  [1553] = {x=-964.119, y=28.121, z=22, rx=180, rz=142.037, shoulder=lefty, elbow=epositive, wrist=wpositive, fatherId=fReference[0]}
  [1554] = {x=-962.88, y=29.088, z=22, rx=180, rz=142.05, shoulder=lefty, elbow=epositive, wrist=wpositive, fatherId=fReference[0]}
  [1555] = {x=-961.641, y=30.054, z=22, rx=180, rz=142.063, shoulder=lefty, elbow=epositive, wrist=wpositive, fatherId=fReference[0]}
  [1556] = {x=-960.402, y=31.02, z=22, rx=180, rz=142.076, shoulder=lefty, elbow=epositive, wrist=wpositive, fatherId=fReference[0]}
  [1557] = {x=-959.163, y=31.986, z=22, rx=180, rz=142.09, shoulder=lefty, elbow=epositive, wrist=wpositive, fatherId=fReference[0]}
  [1558] = {x=-957.923, y=32.951, z=22, rx=180, rz=142.105, shoulder=lefty, elbow=epositive, wrist=wpositive, fatherId=fReference[0]}
  [1559] = {x=-956.684, y=33.916, z=22, rx=180, rz=142.12, shoulder=lefty, elbow=epositive, wrist=wpositive, fatherId=fReference[0]}
  [1560] = {x=-955.444, y=34.88, z=22, rx=180, rz=142.135, shoulder=lefty, elbow=epositive, wrist=wpositive, fatherId=fReference[0]}
  [1561] = {x=-954.204, y=35.844, z=22, rx=180, rz=142.151, shoulder=lefty, elbow=epositive, wrist=wpositive, fatherId=fReference[0]}
  [1562] = {x=-952.964, y=36.808, z=22, rx=180, rz=142.167, shoulder=lefty, elbow=epositive, wrist=wpositive, fatherId=fReference[0]}
  [1563] = {x=-951.724, y=37.771, z=22, rx=180, rz=142.183, shoulder=lefty, elbow=epositive, wrist=wpositive, fatherId=fReference[0]}
  [1564] = {x=-950.483, y=38.734, z=22, rx=180, rz=142.2, shoulder=lefty, elbow=epositive, wrist=wpositive, fatherId=fReference[0]}
  [1565] = {x=-949.243, y=39.696, z=22, rx=180, rz=142.218, shoulder=lefty, elbow=epositive, wrist=wpositive, fatherId=fReference[0]}
  [1566] = {x=-948.002, y=40.658, z=22, rx=180, rz=142.235, shoulder=lefty, elbow=epositive, wrist=wpositive, fatherId=fReference[0]}
  [1567] = {x=-946.761, y=41.619, z=22, rx=180, rz=142.254, shoulder=lefty, elbow=epositive, wrist=wpositive, fatherId=fReference[0]}
  [1568] = {x=-945.52, y=42.58, z=22, rx=180, rz=142.272, shoulder=lefty, elbow=epositive, wrist=wpositive, fatherId=fReference[0]}
  [1569] = {x=-944.278, y=43.541, z=22, rx=180, rz=142.291, shoulder=lefty, elbow=epositive, wrist=wpositive, fatherId=fReference[0]}
  [1570] = {x=-943.037, y=44.501, z=22, rx=180, rz=142.311, shoulder=lefty, elbow=epositive, wrist=wpositive, fatherId=fReference[0]}
  [1571] = {x=-941.795, y=45.46, z=22, rx=180, rz=142.331, shoulder=lefty, elbow=epositive, wrist=wpositive, fatherId=fReference[0]}
  [1572] = {x=-940.553, y=46.419, z=22, rx=180, rz=142.351, shoulder=lefty, elbow=epositive, wrist=wpositive, fatherId=fReference[0]}
  [1573] = {x=-939.31, y=47.377, z=22, rx=180, rz=142.372, shoulder=lefty, elbow=epositive, wrist=wpositive, fatherId=fReference[0]}
  [1574] = {x=-938.068, y=48.335, z=22, rx=180, rz=142.394, shoulder=lefty, elbow=epositive, wrist=wpositive, fatherId=fReference[0]}
  [1575] = {x=-936.825, y=49.292, z=22, rx=180, rz=142.415, shoulder=lefty, elbow=epositive, wrist=wpositive, fatherId=fReference[0]}
  [1576] = {x=-935.582, y=50.249, z=22, rx=180, rz=142.438, shoulder=lefty, elbow=epositive, wrist=wpositive, fatherId=fReference[0]}
  [1577] = {x=-934.339, y=51.205, z=22, rx=180, rz=142.46, shoulder=lefty, elbow=epositive, wrist=wpositive, fatherId=fReference[0]}
  [1578] = {x=-933.095, y=52.161, z=22, rx=180, rz=142.483, shoulder=lefty, elbow=epositive, wrist=wpositive, fatherId=fReference[0]}
  [1579] = {x=-931.852, y=53.116, z=22, rx=180, rz=142.507, shoulder=lefty, elbow=epositive, wrist=wpositive, fatherId=fReference[0]}
  [1580] = {x=-930.608, y=54.07, z=22, rx=180, rz=142.531, shoulder=lefty, elbow=epositive, wrist=wpositive, fatherId=fReference[0]}
  [1581] = {x=-929.363, y=55.024, z=22, rx=180, rz=142.555, shoulder=lefty, elbow=epositive, wrist=wpositive, fatherId=fReference[0]}
  [1582] = {x=-928.119, y=55.977, z=22, rx=180, rz=142.58, shoulder=lefty, elbow=epositive, wrist=wpositive, fatherId=fReference[0]}
  [1583] = {x=-926.874, y=56.929, z=22, rx=180, rz=142.605, shoulder=lefty, elbow=epositive, wrist=wpositive, fatherId=fReference[0]}
  [1584] = {x=-925.629, y=57.881, z=22, rx=180, rz=142.631, shoulder=lefty, elbow=epositive, wrist=wpositive, fatherId=fReference[0]}
  [1585] = {x=-924.384, y=58.832, z=22, rx=180, rz=142.657, shoulder=lefty, elbow=epositive, wrist=wpositive, fatherId=fReference[0]}
  [1586] = {x=-923.138, y=59.782, z=22, rx=180, rz=142.684, shoulder=lefty, elbow=epositive, wrist=wpositive, fatherId=fReference[0]}
  [1587] = {x=-921.892, y=60.732, z=22, rx=180, rz=142.711, shoulder=lefty, elbow=epositive, wrist=wpositive, fatherId=fReference[0]}
  [1588] = {x=-920.646, y=61.681, z=22, rx=180, rz=142.738, shoulder=lefty, elbow=epositive, wrist=wpositive, fatherId=fReference[0]}
  [1589] = {x=-919.4, y=62.629, z=22, rx=180, rz=142.766, shoulder=lefty, elbow=epositive, wrist=wpositive, fatherId=fReference[0]}
  [1590] = {x=-918.153, y=63.576, z=22, rx=180, rz=142.795, shoulder=lefty, elbow=epositive, wrist=wpositive, fatherId=fReference[0]}
  [1591] = {x=-916.906, y=64.523, z=22, rx=180, rz=142.824, shoulder=lefty, elbow=epositive, wrist=wpositive, fatherId=fReference[0]}
  [1592] = {x=-915.659, y=65.469, z=22, rx=180, rz=142.853, shoulder=lefty, elbow=epositive, wrist=wpositive, fatherId=fReference[0]}
  [1593] = {x=-914.411, y=66.414, z=22, rx=180, rz=142.883, shoulder=lefty, elbow=epositive, wrist=wpositive, fatherId=fReference[0]}
  [1594] = {x=-913.163, y=67.358, z=22, rx=180, rz=142.913, shoulder=lefty, elbow=epositive, wrist=wpositive, fatherId=fReference[0]}
  [1595] = {x=-911.915, y=68.302, z=22, rx=180, rz=142.944, shoulder=lefty, elbow=epositive, wrist=wpositive, fatherId=fReference[0]}
  [1596] = {x=-910.667, y=69.245, z=22, rx=180, rz=142.975, shoulder=lefty, elbow=epositive, wrist=wpositive, fatherId=fReference[0]}
  [1597] = {x=-909.418, y=70.187, z=22, rx=180, rz=143.007, shoulder=lefty, elbow=epositive, wrist=wpositive, fatherId=fReference[0]}
  [1598] = {x=-908.169, y=71.128, z=22, rx=180, rz=143.039, shoulder=lefty, elbow=epositive, wrist=wpositive, fatherId=fReference[0]}
  [1599] = {x=-906.919, y=72.068, z=22, rx=180, rz=143.071, shoulder=lefty, elbow=epositive, wrist=wpositive, fatherId=fReference[0]}
  [1600] = {x=-905.67, y=73.007, z=22, rx=180, rz=143.104, shoulder=lefty, elbow=epositive, wrist=wpositive, fatherId=fReference[0]}
  [1601] = {x=-904.419, y=73.946, z=22, rx=180, rz=143.138, shoulder=lefty, elbow=epositive, wrist=wpositive, fatherId=fReference[0]}
  [1602] = {x=-903.169, y=74.883, z=22, rx=180, rz=143.172, shoulder=lefty, elbow=epositive, wrist=wpositive, fatherId=fReference[0]}
  [1603] = {x=-901.918, y=75.82, z=22, rx=180, rz=143.206, shoulder=lefty, elbow=epositive, wrist=wpositive, fatherId=fReference[0]}
  [1604] = {x=-900.667, y=76.756, z=22, rx=180, rz=143.241, shoulder=lefty, elbow=epositive, wrist=wpositive, fatherId=fReference[0]}
  [1605] = {x=-899.416, y=77.691, z=22, rx=180, rz=143.276, shoulder=lefty, elbow=epositive, wrist=wpositive, fatherId=fReference[0]}
  [1606] = {x=-898.164, y=78.625, z=22, rx=180, rz=143.312, shoulder=lefty, elbow=epositive, wrist=wpositive, fatherId=fReference[0]}
  [1607] = {x=-896.912, y=79.557, z=22, rx=180, rz=143.348, shoulder=lefty, elbow=epositive, wrist=wpositive, fatherId=fReference[0]}
  [1608] = {x=-895.659, y=80.489, z=22, rx=180, rz=143.385, shoulder=lefty, elbow=epositive, wrist=wpositive, fatherId=fReference[0]}
  [1609] = {x=-894.406, y=81.42, z=22, rx=180, rz=143.422, shoulder=lefty, elbow=epositive, wrist=wpositive, fatherId=fReference[0]}
  [1610] = {x=-893.153, y=82.35, z=22, rx=180, rz=143.46, shoulder=lefty, elbow=epositive, wrist=wpositive, fatherId=fReference[0]}
  [1611] = {x=-891.899, y=83.279, z=22, rx=180, rz=143.498, shoulder=lefty, elbow=epositive, wrist=wpositive, fatherId=fReference[0]}
  [1612] = {x=-890.645, y=84.207, z=22, rx=180, rz=143.536, shoulder=lefty, elbow=epositive, wrist=wpositive, fatherId=fReference[0]}
  [1613] = {x=-889.391, y=85.134, z=22, rx=180, rz=143.575, shoulder=lefty, elbow=epositive, wrist=wpositive, fatherId=fReference[0]}
  [1614] = {x=-888.136, y=86.06, z=22, rx=180, rz=143.615, shoulder=lefty, elbow=epositive, wrist=wpositive, fatherId=fReference[0]}
  [1615] = {x=-886.881, y=86.985, z=22, rx=180, rz=143.655, shoulder=lefty, elbow=epositive, wrist=wpositive, fatherId=fReference[0]}
  [1616] = {x=-885.626, y=87.909, z=22, rx=180, rz=143.696, shoulder=lefty, elbow=epositive, wrist=wpositive, fatherId=fReference[0]}
  [1617] = {x=-884.37, y=88.832, z=22, rx=180, rz=143.737, shoulder=lefty, elbow=epositive, wrist=wpositive, fatherId=fReference[0]}
  [1618] = {x=-883.113, y=89.753, z=22, rx=180, rz=143.778, shoulder=lefty, elbow=epositive, wrist=wpositive, fatherId=fReference[0]}
  [1619] = {x=-881.857, y=90.674, z=22, rx=180, rz=143.82, shoulder=lefty, elbow=epositive, wrist=wpositive, fatherId=fReference[0]}
  [1620] = {x=-880.6, y=91.593, z=22, rx=180, rz=143.862, shoulder=lefty, elbow=epositive, wrist=wpositive, fatherId=fReference[0]}
  [1621] = {x=-879.342, y=92.511, z=22, rx=180, rz=143.905, shoulder=lefty, elbow=epositive, wrist=wpositive, fatherId=fReference[0]}
  [1622] = {x=-878.084, y=93.428, z=22, rx=180, rz=143.949, shoulder=lefty, elbow=epositive, wrist=wpositive, fatherId=fReference[0]}
  [1623] = {x=-876.826, y=94.344, z=22, rx=180, rz=143.993, shoulder=lefty, elbow=epositive, wrist=wpositive, fatherId=fReference[0]}
  [1624] = {x=-875.567, y=95.259, z=22, rx=180, rz=144.037, shoulder=lefty, elbow=epositive, wrist=wpositive, fatherId=fReference[0]}
  [1625] = {x=-874.308, y=96.173, z=22, rx=180, rz=144.082, shoulder=lefty, elbow=epositive, wrist=wpositive, fatherId=fReference[0]}
  [1626] = {x=-873.049, y=97.085, z=22, rx=180, rz=144.127, shoulder=lefty, elbow=epositive, wrist=wpositive, fatherId=fReference[0]}
  [1627] = {x=-871.789, y=97.996, z=22, rx=180, rz=144.173, shoulder=lefty, elbow=epositive, wrist=wpositive, fatherId=fReference[0]}
  [1628] = {x=-870.528, y=98.906, z=22, rx=-180, rz=144.22, shoulder=lefty, elbow=epositive, wrist=wpositive, fatherId=fReference[0]}
  [1629] = {x=-869.267, y=99.815, z=22, rx=180, rz=144.266, shoulder=lefty, elbow=epositive, wrist=wpositive, fatherId=fReference[0]}
  [1630] = {x=-868.006, y=100.722, z=22, rx=180, rz=144.314, shoulder=lefty, elbow=epositive, wrist=wpositive, fatherId=fReference[0]}
  [1631] = {x=-866.745, y=101.628, z=22, rx=180, rz=144.362, shoulder=lefty, elbow=epositive, wrist=wpositive, fatherId=fReference[0]}
  [1632] = {x=-865.482, y=102.533, z=22, rx=180, rz=144.41, shoulder=lefty, elbow=epositive, wrist=wpositive, fatherId=fReference[0]}
  [1633] = {x=-864.22, y=103.437, z=22, rx=180, rz=144.459, shoulder=lefty, elbow=epositive, wrist=wpositive, fatherId=fReference[0]}
  [1634] = {x=-862.957, y=104.339, z=22, rx=180, rz=144.508, shoulder=lefty, elbow=epositive, wrist=wpositive, fatherId=fReference[0]}
  [1635] = {x=-861.693, y=105.24, z=22, rx=180, rz=144.558, shoulder=lefty, elbow=epositive, wrist=wpositive, fatherId=fReference[0]}
  [1636] = {x=-860.429, y=106.139, z=22, rx=180, rz=144.609, shoulder=lefty, elbow=epositive, wrist=wpositive, fatherId=fReference[0]}
  [1637] = {x=-859.165, y=107.038, z=22, rx=180, rz=144.659, shoulder=lefty, elbow=epositive, wrist=wpositive, fatherId=fReference[0]}
  [1638] = {x=-857.9, y=107.935, z=22, rx=180, rz=144.711, shoulder=lefty, elbow=epositive, wrist=wpositive, fatherId=fReference[0]}
  [1639] = {x=-856.635, y=108.83, z=22, rx=180, rz=144.763, shoulder=lefty, elbow=epositive, wrist=wpositive, fatherId=fReference[0]}
  [1640] = {x=-855.369, y=109.724, z=22, rx=180, rz=144.815, shoulder=lefty, elbow=epositive, wrist=wpositive, fatherId=fReference[0]}
  [1641] = {x=-854.103, y=110.617, z=22, rx=180, rz=144.868, shoulder=lefty, elbow=epositive, wrist=wpositive, fatherId=fReference[0]}
  [1642] = {x=-852.836, y=111.508, z=22, rx=180, rz=144.922, shoulder=lefty, elbow=epositive, wrist=wpositive, fatherId=fReference[0]}
  [1643] = {x=-851.569, y=112.398, z=22, rx=180, rz=144.976, shoulder=lefty, elbow=epositive, wrist=wpositive, fatherId=fReference[0]}
  [1644] = {x=-850.301, y=113.287, z=22, rx=180, rz=145.03, shoulder=lefty, elbow=epositive, wrist=wpositive, fatherId=fReference[0]}
  [1645] = {x=-849.033, y=114.174, z=22, rx=180, rz=145.085, shoulder=lefty, elbow=epositive, wrist=wpositive, fatherId=fReference[0]}
  [1646] = {x=-847.764, y=115.059, z=22, rx=180, rz=145.141, shoulder=lefty, elbow=epositive, wrist=wpositive, fatherId=fReference[0]}
  [1647] = {x=-846.495, y=115.943, z=22, rx=180, rz=145.197, shoulder=lefty, elbow=epositive, wrist=wpositive, fatherId=fReference[0]}
  [1648] = {x=-845.225, y=116.826, z=22, rx=180, rz=145.253, shoulder=lefty, elbow=epositive, wrist=wpositive, fatherId=fReference[0]}
  [1649] = {x=-843.955, y=117.707, z=22, rx=180, rz=145.311, shoulder=lefty, elbow=epositive, wrist=wpositive, fatherId=fReference[0]}
  [1650] = {x=-842.685, y=118.586, z=22, rx=180, rz=145.368, shoulder=lefty, elbow=epositive, wrist=wpositive, fatherId=fReference[0]}
  [1651] = {x=-841.413, y=119.464, z=22, rx=180, rz=145.426, shoulder=lefty, elbow=epositive, wrist=wpositive, fatherId=fReference[0]}
  [1652] = {x=-840.142, y=120.341, z=22, rx=180, rz=145.485, shoulder=lefty, elbow=epositive, wrist=wpositive, fatherId=fReference[0]}
  [1653] = {x=-838.869, y=121.216, z=22, rx=180, rz=145.544, shoulder=lefty, elbow=epositive, wrist=wpositive, fatherId=fReference[0]}
  [1654] = {x=-837.597, y=122.089, z=22, rx=180, rz=145.604, shoulder=lefty, elbow=epositive, wrist=wpositive, fatherId=fReference[0]}
  [1655] = {x=-836.323, y=122.961, z=22, rx=180, rz=145.665, shoulder=lefty, elbow=epositive, wrist=wpositive, fatherId=fReference[0]}
  [1656] = {x=-835.049, y=123.831, z=22, rx=180, rz=145.725, shoulder=lefty, elbow=epositive, wrist=wpositive, fatherId=fReference[0]}
  [1657] = {x=-833.775, y=124.699, z=22, rx=180, rz=145.787, shoulder=lefty, elbow=epositive, wrist=wpositive, fatherId=fReference[0]}
  [1658] = {x=-832.5, y=125.566, z=22, rx=-180, rz=145.849, shoulder=lefty, elbow=epositive, wrist=wpositive, fatherId=fReference[0]}
  [1659] = {x=-831.225, y=126.431, z=22, rx=180, rz=145.911, shoulder=lefty, elbow=epositive, wrist=wpositive, fatherId=fReference[0]}
  [1660] = {x=-829.949, y=127.295, z=22, rx=180, rz=145.974, shoulder=lefty, elbow=epositive, wrist=wpositive, fatherId=fReference[0]}
  [1661] = {x=-828.672, y=128.157, z=22, rx=180, rz=146.038, shoulder=lefty, elbow=epositive, wrist=wpositive, fatherId=fReference[0]}
  [1662] = {x=-827.395, y=129.017, z=22, rx=180, rz=146.102, shoulder=lefty, elbow=epositive, wrist=wpositive, fatherId=fReference[0]}
  [1663] = {x=-826.117, y=129.876, z=22, rx=180, rz=146.167, shoulder=lefty, elbow=epositive, wrist=wpositive, fatherId=fReference[0]}
  [1664] = {x=-824.839, y=130.732, z=22, rx=180, rz=146.232, shoulder=lefty, elbow=epositive, wrist=wpositive, fatherId=fReference[0]}
  [1665] = {x=-823.56, y=131.587, z=22, rx=180, rz=146.298, shoulder=lefty, elbow=epositive, wrist=wpositive, fatherId=fReference[0]}
  [1666] = {x=-822.281, y=132.441, z=22, rx=180, rz=146.364, shoulder=lefty, elbow=epositive, wrist=wpositive, fatherId=fReference[0]}
  [1667] = {x=-821.001, y=133.292, z=22, rx=180, rz=146.431, shoulder=lefty, elbow=epositive, wrist=wpositive, fatherId=fReference[0]}
  [1668] = {x=-819.721, y=134.142, z=22, rx=-180, rz=146.499, shoulder=lefty, elbow=epositive, wrist=wpositive, fatherId=fReference[0]}
  [1669] = {x=-818.44, y=134.99, z=22, rx=180, rz=146.567, shoulder=lefty, elbow=epositive, wrist=wpositive, fatherId=fReference[0]}
  [1670] = {x=-817.158, y=135.836, z=22, rx=180, rz=146.636, shoulder=lefty, elbow=epositive, wrist=wpositive, fatherId=fReference[0]}
  [1671] = {x=-815.876, y=136.68, z=22, rx=180, rz=146.705, shoulder=lefty, elbow=epositive, wrist=wpositive, fatherId=fReference[0]}
  [1672] = {x=-814.593, y=137.523, z=22, rx=180, rz=146.775, shoulder=lefty, elbow=epositive, wrist=wpositive, fatherId=fReference[0]}
  [1673] = {x=-813.309, y=138.364, z=22, rx=180, rz=146.845, shoulder=lefty, elbow=epositive, wrist=wpositive, fatherId=fReference[0]}
  [1674] = {x=-812.025, y=139.202, z=22, rx=180, rz=146.916, shoulder=lefty, elbow=epositive, wrist=wpositive, fatherId=fReference[0]}
  [1675] = {x=-810.74, y=140.039, z=22, rx=180, rz=146.987, shoulder=lefty, elbow=epositive, wrist=wpositive, fatherId=fReference[0]}
  [1676] = {x=-809.455, y=140.875, z=22, rx=180, rz=147.059, shoulder=lefty, elbow=epositive, wrist=wpositive, fatherId=fReference[0]}
  [1677] = {x=-808.169, y=141.708, z=22, rx=180, rz=147.132, shoulder=lefty, elbow=epositive, wrist=wpositive, fatherId=fReference[0]}
  [1678] = {x=-806.883, y=142.539, z=22, rx=180, rz=147.205, shoulder=lefty, elbow=epositive, wrist=wpositive, fatherId=fReference[0]}
  [1679] = {x=-805.596, y=143.368, z=22, rx=180, rz=147.279, shoulder=lefty, elbow=epositive, wrist=wpositive, fatherId=fReference[0]}
  [1680] = {x=-804.308, y=144.196, z=22, rx=180, rz=147.353, shoulder=lefty, elbow=epositive, wrist=wpositive, fatherId=fReference[0]}
  [1681] = {x=-803.019, y=145.021, z=22, rx=180, rz=147.428, shoulder=lefty, elbow=epositive, wrist=wpositive, fatherId=fReference[0]}
  [1682] = {x=-801.73, y=145.845, z=22, rx=-180, rz=147.504, shoulder=lefty, elbow=epositive, wrist=wpositive, fatherId=fReference[0]}
  [1683] = {x=-800.44, y=146.666, z=22, rx=180, rz=147.58, shoulder=lefty, elbow=epositive, wrist=wpositive, fatherId=fReference[0]}
  [1684] = {x=-799.15, y=147.486, z=22, rx=180, rz=147.657, shoulder=lefty, elbow=epositive, wrist=wpositive, fatherId=fReference[0]}
  [1685] = {x=-797.859, y=148.303, z=22, rx=180, rz=147.734, shoulder=lefty, elbow=epositive, wrist=wpositive, fatherId=fReference[0]}
  [1686] = {x=-796.567, y=149.119, z=22, rx=180, rz=147.812, shoulder=lefty, elbow=epositive, wrist=wpositive, fatherId=fReference[0]}
  [1687] = {x=-795.275, y=149.932, z=22, rx=180, rz=147.891, shoulder=lefty, elbow=epositive, wrist=wpositive, fatherId=fReference[0]}
  [1688] = {x=-793.982, y=150.744, z=22, rx=180, rz=147.97, shoulder=lefty, elbow=epositive, wrist=wpositive, fatherId=fReference[0]}
  [1689] = {x=-792.688, y=151.553, z=22, rx=-180, rz=148.05, shoulder=lefty, elbow=epositive, wrist=wpositive, fatherId=fReference[0]}
  [1690] = {x=-791.394, y=152.36, z=22, rx=180, rz=148.13, shoulder=lefty, elbow=epositive, wrist=wpositive, fatherId=fReference[0]}
  [1691] = {x=-790.099, y=153.165, z=22, rx=180, rz=148.211, shoulder=lefty, elbow=epositive, wrist=wpositive, fatherId=fReference[0]}
  [1692] = {x=-788.803, y=153.968, z=22, rx=-180, rz=148.293, shoulder=lefty, elbow=epositive, wrist=wpositive, fatherId=fReference[0]}
  [1693] = {x=-787.507, y=154.769, z=22, rx=180, rz=148.375, shoulder=lefty, elbow=epositive, wrist=wpositive, fatherId=fReference[0]}
  [1694] = {x=-786.21, y=155.568, z=22, rx=180, rz=148.458, shoulder=lefty, elbow=epositive, wrist=wpositive, fatherId=fReference[0]}
  [1695] = {x=-784.912, y=156.365, z=22, rx=180, rz=148.541, shoulder=lefty, elbow=epositive, wrist=wpositive, fatherId=fReference[0]}
  [1696] = {x=-783.613, y=157.159, z=22, rx=-180, rz=148.625, shoulder=lefty, elbow=epositive, wrist=wpositive, fatherId=fReference[0]}
  [1697] = {x=-782.314, y=157.951, z=22, rx=180, rz=148.71, shoulder=lefty, elbow=epositive, wrist=wpositive, fatherId=fReference[0]}
  [1698] = {x=-781.014, y=158.741, z=22, rx=180, rz=148.795, shoulder=lefty, elbow=epositive, wrist=wpositive, fatherId=fReference[0]}
  [1699] = {x=-779.714, y=159.529, z=22, rx=180, rz=148.881, shoulder=lefty, elbow=epositive, wrist=wpositive, fatherId=fReference[0]}
  [1700] = {x=-778.413, y=160.315, z=22, rx=180, rz=148.968, shoulder=lefty, elbow=epositive, wrist=wpositive, fatherId=fReference[0]}
  [1701] = {x=-777.111, y=161.098, z=22, rx=180, rz=149.055, shoulder=lefty, elbow=epositive, wrist=wpositive, fatherId=fReference[0]}
  [1702] = {x=-775.808, y=161.879, z=22, rx=180, rz=149.143, shoulder=lefty, elbow=epositive, wrist=wpositive, fatherId=fReference[0]}
  [1703] = {x=-774.505, y=162.658, z=22, rx=180, rz=149.231, shoulder=lefty, elbow=epositive, wrist=wpositive, fatherId=fReference[0]}
  [1704] = {x=-773.2, y=163.434, z=22, rx=-180, rz=149.32, shoulder=lefty, elbow=epositive, wrist=wpositive, fatherId=fReference[0]}
  [1705] = {x=-771.896, y=164.208, z=22, rx=180, rz=149.41, shoulder=lefty, elbow=epositive, wrist=wpositive, fatherId=fReference[0]}
  [1706] = {x=-770.59, y=164.98, z=22, rx=180, rz=149.5, shoulder=lefty, elbow=epositive, wrist=wpositive, fatherId=fReference[0]}
  [1707] = {x=-769.284, y=165.75, z=22, rx=180, rz=149.591, shoulder=lefty, elbow=epositive, wrist=wpositive, fatherId=fReference[0]}
  [1708] = {x=-767.977, y=166.517, z=22, rx=180, rz=149.683, shoulder=lefty, elbow=epositive, wrist=wpositive, fatherId=fReference[0]}
  [1709] = {x=-766.669, y=167.281, z=22, rx=180, rz=149.775, shoulder=lefty, elbow=epositive, wrist=wpositive, fatherId=fReference[0]}
  [1710] = {x=-765.36, y=168.044, z=22, rx=180, rz=149.868, shoulder=lefty, elbow=epositive, wrist=wpositive, fatherId=fReference[0]}
  [1711] = {x=-764.051, y=168.804, z=22, rx=180, rz=149.962, shoulder=lefty, elbow=epositive, wrist=wpositive, fatherId=fReference[0]}
  [1712] = {x=-762.741, y=169.561, z=22, rx=180, rz=150.056, shoulder=lefty, elbow=epositive, wrist=wpositive, fatherId=fReference[0]}
  [1713] = {x=-761.431, y=170.316, z=22, rx=-180, rz=150.151, shoulder=lefty, elbow=epositive, wrist=wpositive, fatherId=fReference[0]}
  [1714] = {x=-760.119, y=171.069, z=22, rx=180, rz=150.247, shoulder=lefty, elbow=epositive, wrist=wpositive, fatherId=fReference[0]}
  [1715] = {x=-758.807, y=171.819, z=22, rx=180, rz=150.343, shoulder=lefty, elbow=epositive, wrist=wpositive, fatherId=fReference[0]}
  [1716] = {x=-757.494, y=172.566, z=22, rx=-180, rz=150.44, shoulder=lefty, elbow=epositive, wrist=wpositive, fatherId=fReference[0]}
  [1717] = {x=-756.181, y=173.311, z=22, rx=180, rz=150.537, shoulder=lefty, elbow=epositive, wrist=wpositive, fatherId=fReference[0]}
  [1718] = {x=-754.866, y=174.054, z=22, rx=180, rz=150.636, shoulder=lefty, elbow=epositive, wrist=wpositive, fatherId=fReference[0]}
  [1719] = {x=-753.551, y=174.794, z=22, rx=180, rz=150.734, shoulder=lefty, elbow=epositive, wrist=wpositive, fatherId=fReference[0]}
  [1720] = {x=-752.235, y=175.531, z=22, rx=180, rz=150.834, shoulder=lefty, elbow=epositive, wrist=wpositive, fatherId=fReference[0]}
  [1721] = {x=-750.919, y=176.266, z=22, rx=180, rz=150.934, shoulder=lefty, elbow=epositive, wrist=wpositive, fatherId=fReference[0]}
  [1722] = {x=-749.601, y=176.998, z=22, rx=180, rz=151.035, shoulder=lefty, elbow=epositive, wrist=wpositive, fatherId=fReference[0]}
  [1723] = {x=-748.283, y=177.727, z=22, rx=180, rz=151.137, shoulder=lefty, elbow=epositive, wrist=wpositive, fatherId=fReference[0]}
  [1724] = {x=-746.965, y=178.454, z=22, rx=180, rz=151.239, shoulder=lefty, elbow=epositive, wrist=wpositive, fatherId=fReference[0]}
  [1725] = {x=-745.645, y=179.179, z=22, rx=180, rz=151.342, shoulder=lefty, elbow=epositive, wrist=wpositive, fatherId=fReference[0]}
  [1726] = {x=-744.325, y=179.9, z=22, rx=180, rz=151.445, shoulder=lefty, elbow=epositive, wrist=wpositive, fatherId=fReference[0]}
  [1727] = {x=-743.004, y=180.619, z=22, rx=180, rz=151.549, shoulder=lefty, elbow=epositive, wrist=wpositive, fatherId=fReference[0]}
  [1728] = {x=-741.682, y=181.335, z=22, rx=180, rz=151.654, shoulder=lefty, elbow=epositive, wrist=wpositive, fatherId=fReference[0]}
  [1729] = {x=-740.359, y=182.049, z=22, rx=180, rz=151.76, shoulder=lefty, elbow=epositive, wrist=wpositive, fatherId=fReference[0]}
  [1730] = {x=-739.036, y=182.76, z=22, rx=180, rz=151.866, shoulder=lefty, elbow=epositive, wrist=wpositive, fatherId=fReference[0]}
  [1731] = {x=-737.712, y=183.468, z=22, rx=-180, rz=151.973, shoulder=lefty, elbow=epositive, wrist=wpositive, fatherId=fReference[0]}
  [1732] = {x=-736.387, y=184.173, z=22, rx=-180, rz=152.081, shoulder=lefty, elbow=epositive, wrist=wpositive, fatherId=fReference[0]}
  [1733] = {x=-735.061, y=184.875, z=22, rx=180, rz=152.189, shoulder=lefty, elbow=epositive, wrist=wpositive, fatherId=fReference[0]}
  [1734] = {x=-733.735, y=185.575, z=22, rx=180, rz=152.298, shoulder=lefty, elbow=epositive, wrist=wpositive, fatherId=fReference[0]}
  [1735] = {x=-732.408, y=186.272, z=22, rx=180, rz=152.408, shoulder=lefty, elbow=epositive, wrist=wpositive, fatherId=fReference[0]}
  [1736] = {x=-731.08, y=186.966, z=22, rx=-180, rz=152.518, shoulder=lefty, elbow=epositive, wrist=wpositive, fatherId=fReference[0]}
  [1737] = {x=-729.751, y=187.657, z=22, rx=180, rz=152.63, shoulder=lefty, elbow=epositive, wrist=wpositive, fatherId=fReference[0]}
  [1738] = {x=-728.422, y=188.345, z=22, rx=-180, rz=152.741, shoulder=lefty, elbow=epositive, wrist=wpositive, fatherId=fReference[0]}
  [1739] = {x=-727.092, y=189.03, z=22, rx=180, rz=152.854, shoulder=lefty, elbow=epositive, wrist=wpositive, fatherId=fReference[0]}
  [1740] = {x=-725.761, y=189.713, z=22, rx=180, rz=152.967, shoulder=lefty, elbow=epositive, wrist=wpositive, fatherId=fReference[0]}
  [1741] = {x=-724.429, y=190.392, z=22, rx=180, rz=153.081, shoulder=lefty, elbow=epositive, wrist=wpositive, fatherId=fReference[0]}
  [1742] = {x=-723.097, y=191.069, z=22, rx=180, rz=153.196, shoulder=lefty, elbow=epositive, wrist=wpositive, fatherId=fReference[0]}
  [1743] = {x=-721.764, y=191.742, z=22, rx=180, rz=153.311, shoulder=lefty, elbow=epositive, wrist=wpositive, fatherId=fReference[0]}
  [1744] = {x=-720.43, y=192.413, z=22, rx=180, rz=153.427, shoulder=lefty, elbow=epositive, wrist=wpositive, fatherId=fReference[0]}
  [1745] = {x=-719.095, y=193.08, z=22, rx=180, rz=153.544, shoulder=lefty, elbow=epositive, wrist=wpositive, fatherId=fReference[0]}
  [1746] = {x=-717.76, y=193.745, z=22, rx=180, rz=153.661, shoulder=lefty, elbow=epositive, wrist=wpositive, fatherId=fReference[0]}
  [1747] = {x=-716.424, y=194.406, z=22, rx=-180, rz=153.779, shoulder=lefty, elbow=epositive, wrist=wpositive, fatherId=fReference[0]}
  [1748] = {x=-715.087, y=195.065, z=22, rx=180, rz=153.898, shoulder=lefty, elbow=epositive, wrist=wpositive, fatherId=fReference[0]}
  [1749] = {x=-713.749, y=195.72, z=22, rx=180, rz=154.017, shoulder=lefty, elbow=epositive, wrist=wpositive, fatherId=fReference[0]}
  [1750] = {x=-712.411, y=196.372, z=22, rx=180, rz=154.138, shoulder=lefty, elbow=epositive, wrist=wpositive, fatherId=fReference[0]}
  [1751] = {x=-711.072, y=197.022, z=22, rx=180, rz=154.259, shoulder=lefty, elbow=epositive, wrist=wpositive, fatherId=fReference[0]}
  [1752] = {x=-709.732, y=197.668, z=22, rx=-180, rz=154.38, shoulder=lefty, elbow=epositive, wrist=wpositive, fatherId=fReference[0]}
  [1753] = {x=-708.391, y=198.311, z=22, rx=180, rz=154.503, shoulder=lefty, elbow=epositive, wrist=wpositive, fatherId=fReference[0]}
  [1754] = {x=-707.05, y=198.95, z=22, rx=180, rz=154.626, shoulder=lefty, elbow=epositive, wrist=wpositive, fatherId=fReference[0]}
  [1755] = {x=-705.708, y=199.587, z=22, rx=180, rz=154.75, shoulder=lefty, elbow=epositive, wrist=wpositive, fatherId=fReference[0]}
  [1756] = {x=-704.365, y=200.22, z=22, rx=-180, rz=154.874, shoulder=lefty, elbow=epositive, wrist=wpositive, fatherId=fReference[0]}
  [1757] = {x=-703.021, y=200.85, z=22, rx=-180, rz=154.999, shoulder=lefty, elbow=epositive, wrist=wpositive, fatherId=fReference[0]}
  [1758] = {x=-701.677, y=201.477, z=22, rx=180, rz=155.125, shoulder=lefty, elbow=epositive, wrist=wpositive, fatherId=fReference[0]}
  [1759] = {x=-700.332, y=202.101, z=22, rx=-180, rz=155.252, shoulder=lefty, elbow=epositive, wrist=wpositive, fatherId=fReference[0]}
  [1760] = {x=-698.986, y=202.721, z=22, rx=180, rz=155.379, shoulder=lefty, elbow=epositive, wrist=wpositive, fatherId=fReference[0]}
  [1761] = {x=-697.639, y=203.338, z=22, rx=180, rz=155.508, shoulder=lefty, elbow=epositive, wrist=wpositive, fatherId=fReference[0]}
  [1762] = {x=-696.292, y=203.952, z=22, rx=180, rz=155.636, shoulder=lefty, elbow=epositive, wrist=wpositive, fatherId=fReference[0]}
  [1763] = {x=-694.944, y=204.563, z=22, rx=180, rz=155.766, shoulder=lefty, elbow=epositive, wrist=wpositive, fatherId=fReference[0]}
  [1764] = {x=-693.595, y=205.17, z=22, rx=180, rz=155.896, shoulder=lefty, elbow=epositive, wrist=wpositive, fatherId=fReference[0]}
  [1765] = {x=-692.246, y=205.774, z=22, rx=180, rz=156.027, shoulder=lefty, elbow=epositive, wrist=wpositive, fatherId=fReference[0]}
  [1766] = {x=-690.895, y=206.374, z=22, rx=180, rz=156.159, shoulder=lefty, elbow=epositive, wrist=wpositive, fatherId=fReference[0]}
  [1767] = {x=-689.544, y=206.971, z=22, rx=180, rz=156.291, shoulder=lefty, elbow=epositive, wrist=wpositive, fatherId=fReference[0]}
  [1768] = {x=-688.193, y=207.565, z=22, rx=180, rz=156.425, shoulder=lefty, elbow=epositive, wrist=wpositive, fatherId=fReference[0]}
  [1769] = {x=-686.84, y=208.155, z=22, rx=180, rz=156.559, shoulder=lefty, elbow=epositive, wrist=wpositive, fatherId=fReference[0]}
  [1770] = {x=-685.487, y=208.741, z=22, rx=180, rz=156.693, shoulder=lefty, elbow=epositive, wrist=wpositive, fatherId=fReference[0]}
  [1771] = {x=-684.133, y=209.325, z=22, rx=-180, rz=156.828, shoulder=lefty, elbow=epositive, wrist=wpositive, fatherId=fReference[0]}
  [1772] = {x=-682.778, y=209.905, z=22, rx=180, rz=156.965, shoulder=lefty, elbow=epositive, wrist=wpositive, fatherId=fReference[0]}
  [1773] = {x=-681.423, y=210.481, z=22, rx=180, rz=157.101, shoulder=lefty, elbow=epositive, wrist=wpositive, fatherId=fReference[0]}
  [1774] = {x=-680.067, y=211.054, z=22, rx=180, rz=157.239, shoulder=lefty, elbow=epositive, wrist=wpositive, fatherId=fReference[0]}
  [1775] = {x=-678.71, y=211.623, z=22, rx=180, rz=157.377, shoulder=lefty, elbow=epositive, wrist=wpositive, fatherId=fReference[0]}
  [1776] = {x=-677.353, y=212.189, z=22, rx=180, rz=157.516, shoulder=lefty, elbow=epositive, wrist=wpositive, fatherId=fReference[0]}
  [1777] = {x=-675.994, y=212.751, z=22, rx=180, rz=157.656, shoulder=lefty, elbow=epositive, wrist=wpositive, fatherId=fReference[0]}
  [1778] = {x=-674.635, y=213.309, z=22, rx=180, rz=157.796, shoulder=lefty, elbow=epositive, wrist=wpositive, fatherId=fReference[0]}
  [1779] = {x=-673.276, y=213.864, z=22, rx=180, rz=157.937, shoulder=lefty, elbow=epositive, wrist=wpositive, fatherId=fReference[0]}
  [1780] = {x=-671.915, y=214.416, z=22, rx=180, rz=158.079, shoulder=lefty, elbow=epositive, wrist=wpositive, fatherId=fReference[0]}
  [1781] = {x=-670.554, y=214.963, z=22, rx=180, rz=158.222, shoulder=lefty, elbow=epositive, wrist=wpositive, fatherId=fReference[0]}
  [1782] = {x=-669.193, y=215.508, z=22, rx=-180, rz=158.365, shoulder=lefty, elbow=epositive, wrist=wpositive, fatherId=fReference[0]}
  [1783] = {x=-667.83, y=216.048, z=22, rx=180, rz=158.509, shoulder=lefty, elbow=epositive, wrist=wpositive, fatherId=fReference[0]}
  [1784] = {x=-666.467, y=216.585, z=22, rx=-180, rz=158.654, shoulder=lefty, elbow=epositive, wrist=wpositive, fatherId=fReference[0]}
  [1785] = {x=-665.103, y=217.118, z=22, rx=180, rz=158.799, shoulder=lefty, elbow=epositive, wrist=wpositive, fatherId=fReference[0]}
  [1786] = {x=-663.739, y=217.647, z=22, rx=180, rz=158.945, shoulder=lefty, elbow=epositive, wrist=wpositive, fatherId=fReference[0]}
  [1787] = {x=-662.373, y=218.173, z=22, rx=180, rz=159.092, shoulder=lefty, elbow=epositive, wrist=wpositive, fatherId=fReference[0]}
  [1788] = {x=-661.007, y=218.694, z=22, rx=180, rz=159.24, shoulder=lefty, elbow=epositive, wrist=wpositive, fatherId=fReference[0]}
  [1789] = {x=-659.641, y=219.212, z=22, rx=-180, rz=159.388, shoulder=lefty, elbow=epositive, wrist=wpositive, fatherId=fReference[0]}
  [1790] = {x=-658.273, y=219.727, z=22, rx=180, rz=159.537, shoulder=lefty, elbow=epositive, wrist=wpositive, fatherId=fReference[0]}
  [1791] = {x=-656.905, y=220.237, z=22, rx=180, rz=159.687, shoulder=lefty, elbow=epositive, wrist=wpositive, fatherId=fReference[0]}
  [1792] = {x=-655.537, y=220.744, z=22, rx=180, rz=159.837, shoulder=lefty, elbow=epositive, wrist=wpositive, fatherId=fReference[0]}
  [1793] = {x=-654.167, y=221.247, z=22, rx=180, rz=159.988, shoulder=lefty, elbow=epositive, wrist=wpositive, fatherId=fReference[0]}
  [1794] = {x=-652.797, y=221.746, z=22, rx=180, rz=160.14, shoulder=lefty, elbow=epositive, wrist=wpositive, fatherId=fReference[0]}
  [1795] = {x=-651.426, y=222.241, z=22, rx=180, rz=160.293, shoulder=lefty, elbow=epositive, wrist=wpositive, fatherId=fReference[0]}
  [1796] = {x=-650.055, y=222.732, z=22, rx=180, rz=160.446, shoulder=lefty, elbow=epositive, wrist=wpositive, fatherId=fReference[0]}
  [1797] = {x=-648.683, y=223.219, z=22, rx=180, rz=160.6, shoulder=lefty, elbow=epositive, wrist=wpositive, fatherId=fReference[0]}
  [1798] = {x=-647.31, y=223.703, z=22, rx=180, rz=160.755, shoulder=lefty, elbow=epositive, wrist=wpositive, fatherId=fReference[0]}
  [1799] = {x=-645.937, y=224.182, z=22, rx=180, rz=160.91, shoulder=lefty, elbow=epositive, wrist=wpositive, fatherId=fReference[0]}
  [1800] = {x=-644.562, y=224.658, z=22, rx=180, rz=161.066, shoulder=lefty, elbow=epositive, wrist=wpositive, fatherId=fReference[0]}
  [1801] = {x=-643.188, y=225.129, z=22, rx=-180, rz=161.223, shoulder=lefty, elbow=epositive, wrist=wpositive, fatherId=fReference[0]}
  [1802] = {x=-641.812, y=225.597, z=22, rx=180, rz=161.381, shoulder=lefty, elbow=epositive, wrist=wpositive, fatherId=fReference[0]}
  [1803] = {x=-640.436, y=226.061, z=22, rx=-180, rz=161.539, shoulder=lefty, elbow=epositive, wrist=wpositive, fatherId=fReference[0]}
  [1804] = {x=-639.06, y=226.52, z=22, rx=180, rz=161.698, shoulder=lefty, elbow=epositive, wrist=wpositive, fatherId=fReference[0]}
  [1805] = {x=-637.682, y=226.976, z=22, rx=180, rz=161.857, shoulder=lefty, elbow=epositive, wrist=wpositive, fatherId=fReference[0]}
  [1806] = {x=-636.304, y=227.427, z=22, rx=180, rz=162.017, shoulder=lefty, elbow=epositive, wrist=wpositive, fatherId=fReference[0]}
  [1807] = {x=-634.925, y=227.875, z=22, rx=180, rz=162.178, shoulder=lefty, elbow=epositive, wrist=wpositive, fatherId=fReference[0]}
  [1808] = {x=-633.546, y=228.318, z=22, rx=-180, rz=162.34, shoulder=lefty, elbow=epositive, wrist=wpositive, fatherId=fReference[0]}
  [1809] = {x=-632.166, y=228.758, z=22, rx=180, rz=162.502, shoulder=lefty, elbow=epositive, wrist=wpositive, fatherId=fReference[0]}
  [1810] = {x=-630.786, y=229.193, z=22, rx=-180, rz=162.665, shoulder=lefty, elbow=epositive, wrist=wpositive, fatherId=fReference[0]}
  [1811] = {x=-629.404, y=229.624, z=22, rx=180, rz=162.829, shoulder=lefty, elbow=epositive, wrist=wpositive, fatherId=fReference[0]}
  [1812] = {x=-628.022, y=230.051, z=22, rx=180, rz=162.993, shoulder=lefty, elbow=epositive, wrist=wpositive, fatherId=fReference[0]}
  [1813] = {x=-626.64, y=230.474, z=22, rx=180, rz=163.158, shoulder=lefty, elbow=epositive, wrist=wpositive, fatherId=fReference[0]}
  [1814] = {x=-625.257, y=230.893, z=22, rx=180, rz=163.324, shoulder=lefty, elbow=epositive, wrist=wpositive, fatherId=fReference[0]}
  [1815] = {x=-623.873, y=231.307, z=22, rx=180, rz=163.49, shoulder=lefty, elbow=epositive, wrist=wpositive, fatherId=fReference[0]}
  [1816] = {x=-622.489, y=231.717, z=22, rx=-180, rz=163.657, shoulder=lefty, elbow=epositive, wrist=wpositive, fatherId=fReference[0]}
  [1817] = {x=-621.104, y=232.124, z=22, rx=180, rz=163.824, shoulder=lefty, elbow=epositive, wrist=wpositive, fatherId=fReference[0]}
  [1818] = {x=-619.718, y=232.526, z=22, rx=180, rz=163.993, shoulder=lefty, elbow=epositive, wrist=wpositive, fatherId=fReference[0]}
  [1819] = {x=-618.332, y=232.923, z=22, rx=180, rz=164.161, shoulder=lefty, elbow=epositive, wrist=wpositive, fatherId=fReference[0]}
  [1820] = {x=-616.945, y=233.317, z=22, rx=180, rz=164.331, shoulder=lefty, elbow=epositive, wrist=wpositive, fatherId=fReference[0]}
  [1821] = {x=-615.558, y=233.706, z=22, rx=180, rz=164.501, shoulder=lefty, elbow=epositive, wrist=wpositive, fatherId=fReference[0]}
  [1822] = {x=-614.17, y=234.091, z=22, rx=180, rz=164.672, shoulder=lefty, elbow=epositive, wrist=wpositive, fatherId=fReference[0]}
  [1823] = {x=-612.781, y=234.471, z=22, rx=180, rz=164.843, shoulder=lefty, elbow=epositive, wrist=wpositive, fatherId=fReference[0]}
  [1824] = {x=-611.392, y=234.848, z=22, rx=-180, rz=165.015, shoulder=lefty, elbow=epositive, wrist=wpositive, fatherId=fReference[0]}
  [1825] = {x=-610.002, y=235.22, z=22, rx=180, rz=165.188, shoulder=lefty, elbow=epositive, wrist=wpositive, fatherId=fReference[0]}
  [1826] = {x=-608.612, y=235.587, z=22, rx=180, rz=165.361, shoulder=lefty, elbow=epositive, wrist=wpositive, fatherId=fReference[0]}
  [1827] = {x=-607.221, y=235.951, z=22, rx=180, rz=165.535, shoulder=lefty, elbow=epositive, wrist=wpositive, fatherId=fReference[0]}
  [1828] = {x=-605.829, y=236.31, z=22, rx=180, rz=165.71, shoulder=lefty, elbow=epositive, wrist=wpositive, fatherId=fReference[0]}
  [1829] = {x=-604.437, y=236.664, z=22, rx=-180, rz=165.885, shoulder=lefty, elbow=epositive, wrist=wpositive, fatherId=fReference[0]}
  [1830] = {x=-603.045, y=237.014, z=22, rx=-180, rz=166.061, shoulder=lefty, elbow=epositive, wrist=wpositive, fatherId=fReference[0]}
  [1831] = {x=-601.652, y=237.36, z=22, rx=180, rz=166.237, shoulder=lefty, elbow=epositive, wrist=wpositive, fatherId=fReference[0]}
  [1832] = {x=-600.258, y=237.701, z=22, rx=-180, rz=166.414, shoulder=lefty, elbow=epositive, wrist=wpositive, fatherId=fReference[0]}
  [1833] = {x=-598.864, y=238.038, z=22, rx=-180, rz=166.591, shoulder=lefty, elbow=epositive, wrist=wpositive, fatherId=fReference[0]}
  [1834] = {x=-597.469, y=238.371, z=22, rx=-180, rz=166.77, shoulder=lefty, elbow=epositive, wrist=wpositive, fatherId=fReference[0]}
  [1835] = {x=-596.074, y=238.699, z=22, rx=-180, rz=166.948, shoulder=lefty, elbow=epositive, wrist=wpositive, fatherId=fReference[0]}
  [1836] = {x=-594.678, y=239.023, z=22, rx=180, rz=167.127, shoulder=lefty, elbow=epositive, wrist=wpositive, fatherId=fReference[0]}
  [1837] = {x=-593.281, y=239.342, z=22, rx=180, rz=167.307, shoulder=lefty, elbow=epositive, wrist=wpositive, fatherId=fReference[0]}
  [1838] = {x=-591.885, y=239.656, z=22, rx=-180, rz=167.487, shoulder=lefty, elbow=epositive, wrist=wpositive, fatherId=fReference[0]}
  [1839] = {x=-590.487, y=239.966, z=22, rx=180, rz=167.668, shoulder=lefty, elbow=epositive, wrist=wpositive, fatherId=fReference[0]}
  [1840] = {x=-589.09, y=240.272, z=22, rx=180, rz=167.85, shoulder=lefty, elbow=epositive, wrist=wpositive, fatherId=fReference[0]}
  [1841] = {x=-587.691, y=240.573, z=22, rx=180, rz=168.032, shoulder=lefty, elbow=epositive, wrist=wpositive, fatherId=fReference[0]}
  [1842] = {x=-586.292, y=240.869, z=22, rx=180, rz=168.214, shoulder=lefty, elbow=epositive, wrist=wpositive, fatherId=fReference[0]}
  [1843] = {x=-584.893, y=241.161, z=22, rx=180, rz=168.397, shoulder=lefty, elbow=epositive, wrist=wpositive, fatherId=fReference[0]}
  [1844] = {x=-583.493, y=241.449, z=22, rx=180, rz=168.581, shoulder=lefty, elbow=epositive, wrist=wpositive, fatherId=fReference[0]}
  [1845] = {x=-582.093, y=241.732, z=22, rx=-180, rz=168.765, shoulder=lefty, elbow=epositive, wrist=wpositive, fatherId=fReference[0]}
  [1846] = {x=-580.693, y=242.01, z=22, rx=-180, rz=168.949, shoulder=lefty, elbow=epositive, wrist=wpositive, fatherId=fReference[0]}
  [1847] = {x=-579.292, y=242.283, z=22, rx=180, rz=169.134, shoulder=lefty, elbow=epositive, wrist=wpositive, fatherId=fReference[0]}
  [1848] = {x=-577.89, y=242.553, z=22, rx=180, rz=169.32, shoulder=lefty, elbow=epositive, wrist=wpositive, fatherId=fReference[0]}
  [1849] = {x=-576.488, y=242.817, z=22, rx=180, rz=169.506, shoulder=lefty, elbow=epositive, wrist=wpositive, fatherId=fReference[0]}
  [1850] = {x=-575.086, y=243.077, z=22, rx=180, rz=169.692, shoulder=lefty, elbow=epositive, wrist=wpositive, fatherId=fReference[0]}
  [1851] = {x=-573.683, y=243.332, z=22, rx=180, rz=169.879, shoulder=lefty, elbow=epositive, wrist=wpositive, fatherId=fReference[0]}
  [1852] = {x=-572.279, y=243.582, z=22, rx=-180, rz=170.067, shoulder=lefty, elbow=epositive, wrist=wpositive, fatherId=fReference[0]}
  [1853] = {x=-570.876, y=243.828, z=22, rx=180, rz=170.255, shoulder=lefty, elbow=epositive, wrist=wpositive, fatherId=fReference[0]}
  [1854] = {x=-569.472, y=244.069, z=22, rx=-180, rz=170.443, shoulder=lefty, elbow=epositive, wrist=wpositive, fatherId=fReference[0]}
  [1855] = {x=-568.067, y=244.306, z=22, rx=-180, rz=170.632, shoulder=lefty, elbow=epositive, wrist=wpositive, fatherId=fReference[0]}
  [1856] = {x=-566.662, y=244.538, z=22, rx=-180, rz=170.821, shoulder=lefty, elbow=epositive, wrist=wpositive, fatherId=fReference[0]}
  [1857] = {x=-565.257, y=244.765, z=22, rx=-180, rz=171.011, shoulder=lefty, elbow=epositive, wrist=wpositive, fatherId=fReference[0]}
  [1858] = {x=-563.852, y=244.987, z=22, rx=180, rz=171.201, shoulder=lefty, elbow=epositive, wrist=wpositive, fatherId=fReference[0]}
  [1859] = {x=-562.446, y=245.205, z=22, rx=180, rz=171.391, shoulder=lefty, elbow=epositive, wrist=wpositive, fatherId=fReference[0]}
  [1860] = {x=-561.039, y=245.417, z=22, rx=180, rz=171.582, shoulder=lefty, elbow=epositive, wrist=wpositive, fatherId=fReference[0]}
  [1861] = {x=-559.632, y=245.626, z=22, rx=-180, rz=171.774, shoulder=lefty, elbow=epositive, wrist=wpositive, fatherId=fReference[0]}
  [1862] = {x=-558.225, y=245.829, z=22, rx=180, rz=171.965, shoulder=lefty, elbow=epositive, wrist=wpositive, fatherId=fReference[0]}
  [1863] = {x=-556.818, y=246.028, z=22, rx=180, rz=172.157, shoulder=lefty, elbow=epositive, wrist=wpositive, fatherId=fReference[0]}
  [1864] = {x=-555.41, y=246.222, z=22, rx=180, rz=172.35, shoulder=lefty, elbow=epositive, wrist=wpositive, fatherId=fReference[0]}
  [1865] = {x=-554.002, y=246.411, z=22, rx=180, rz=172.543, shoulder=lefty, elbow=epositive, wrist=wpositive, fatherId=fReference[0]}
  [1866] = {x=-552.594, y=246.595, z=22, rx=180, rz=172.736, shoulder=lefty, elbow=epositive, wrist=wpositive, fatherId=fReference[0]}
  [1867] = {x=-551.185, y=246.775, z=22, rx=-180, rz=172.929, shoulder=lefty, elbow=epositive, wrist=wpositive, fatherId=fReference[0]}
  [1868] = {x=-549.776, y=246.949, z=22, rx=-180, rz=173.123, shoulder=lefty, elbow=epositive, wrist=wpositive, fatherId=fReference[0]}
  [1869] = {x=-548.367, y=247.119, z=22, rx=180, rz=173.317, shoulder=lefty, elbow=epositive, wrist=wpositive, fatherId=fReference[0]}
  [1870] = {x=-546.957, y=247.285, z=22, rx=180, rz=173.512, shoulder=lefty, elbow=epositive, wrist=wpositive, fatherId=fReference[0]}
  [1871] = {x=-545.548, y=247.445, z=22, rx=180, rz=173.707, shoulder=lefty, elbow=epositive, wrist=wpositive, fatherId=fReference[0]}
  [1872] = {x=-544.137, y=247.6, z=22, rx=180, rz=173.902, shoulder=lefty, elbow=epositive, wrist=wpositive, fatherId=fReference[0]}
  [1873] = {x=-542.727, y=247.751, z=22, rx=180, rz=174.097, shoulder=lefty, elbow=epositive, wrist=wpositive, fatherId=fReference[0]}
  [1874] = {x=-541.316, y=247.897, z=22, rx=180, rz=174.293, shoulder=lefty, elbow=epositive, wrist=wpositive, fatherId=fReference[0]}
  [1875] = {x=-539.905, y=248.038, z=22, rx=180, rz=174.489, shoulder=lefty, elbow=epositive, wrist=wpositive, fatherId=fReference[0]}
  [1876] = {x=-538.494, y=248.174, z=22, rx=-180, rz=174.685, shoulder=lefty, elbow=epositive, wrist=wpositive, fatherId=fReference[0]}
  [1877] = {x=-537.083, y=248.305, z=22, rx=-180, rz=174.882, shoulder=lefty, elbow=epositive, wrist=wpositive, fatherId=fReference[0]}
  [1878] = {x=-535.671, y=248.432, z=22, rx=180, rz=175.079, shoulder=lefty, elbow=epositive, wrist=wpositive, fatherId=fReference[0]}
  [1879] = {x=-534.26, y=248.553, z=22, rx=180, rz=175.276, shoulder=lefty, elbow=epositive, wrist=wpositive, fatherId=fReference[0]}
  [1880] = {x=-532.848, y=248.67, z=22, rx=-180, rz=175.473, shoulder=lefty, elbow=epositive, wrist=wpositive, fatherId=fReference[0]}
  [1881] = {x=-531.435, y=248.782, z=22, rx=180, rz=175.671, shoulder=lefty, elbow=epositive, wrist=wpositive, fatherId=fReference[0]}
  [1882] = {x=-530.023, y=248.889, z=22, rx=-180, rz=175.868, shoulder=lefty, elbow=epositive, wrist=wpositive, fatherId=fReference[0]}
  [1883] = {x=-528.61, y=248.991, z=22, rx=-180, rz=176.066, shoulder=lefty, elbow=epositive, wrist=wpositive, fatherId=fReference[0]}
  [1884] = {x=-527.198, y=249.088, z=22, rx=180, rz=176.264, shoulder=lefty, elbow=epositive, wrist=wpositive, fatherId=fReference[0]}
  [1885] = {x=-525.785, y=249.18, z=22, rx=-180, rz=176.463, shoulder=lefty, elbow=epositive, wrist=wpositive, fatherId=fReference[0]}
  [1886] = {x=-524.372, y=249.268, z=22, rx=180, rz=176.661, shoulder=lefty, elbow=epositive, wrist=wpositive, fatherId=fReference[0]}
  [1887] = {x=-522.958, y=249.35, z=22, rx=180, rz=176.86, shoulder=lefty, elbow=epositive, wrist=wpositive, fatherId=fReference[0]}
  [1888] = {x=-521.545, y=249.428, z=22, rx=180, rz=177.059, shoulder=lefty, elbow=epositive, wrist=wpositive, fatherId=fReference[0]}
  [1889] = {x=-520.132, y=249.5, z=22, rx=180, rz=177.258, shoulder=lefty, elbow=epositive, wrist=wpositive, fatherId=fReference[0]}
  [1890] = {x=-518.718, y=249.568, z=22, rx=-180, rz=177.457, shoulder=lefty, elbow=epositive, wrist=wpositive, fatherId=fReference[0]}
  [1891] = {x=-517.304, y=249.631, z=22, rx=180, rz=177.656, shoulder=lefty, elbow=epositive, wrist=wpositive, fatherId=fReference[0]}
  [1892] = {x=-515.89, y=249.689, z=22, rx=-180, rz=177.855, shoulder=lefty, elbow=epositive, wrist=wpositive, fatherId=fReference[0]}
  [1893] = {x=-514.476, y=249.742, z=22, rx=180, rz=178.055, shoulder=lefty, elbow=epositive, wrist=wpositive, fatherId=fReference[0]}
  [1894] = {x=-513.062, y=249.79, z=22, rx=-180, rz=178.254, shoulder=lefty, elbow=epositive, wrist=wpositive, fatherId=fReference[0]}
  [1895] = {x=-511.648, y=249.833, z=22, rx=180, rz=178.454, shoulder=lefty, elbow=epositive, wrist=wpositive, fatherId=fReference[0]}
  [1896] = {x=-510.234, y=249.871, z=22, rx=-180, rz=178.654, shoulder=lefty, elbow=epositive, wrist=wpositive, fatherId=fReference[0]}
  [1897] = {x=-508.82, y=249.904, z=22, rx=180, rz=178.853, shoulder=lefty, elbow=epositive, wrist=wpositive, fatherId=fReference[0]}
  [1898] = {x=-507.405, y=249.932, z=22, rx=180, rz=179.053, shoulder=lefty, elbow=epositive, wrist=wpositive, fatherId=fReference[0]}
  [1899] = {x=-505.991, y=249.956, z=22, rx=-180, rz=179.253, shoulder=lefty, elbow=epositive, wrist=wpositive, fatherId=fReference[0]}
  [1900] = {x=-504.577, y=249.974, z=22, rx=180, rz=179.453, shoulder=lefty, elbow=epositive, wrist=wpositive, fatherId=fReference[0]}
  [1901] = {x=-503.162, y=249.988, z=22, rx=180, rz=179.653, shoulder=lefty, elbow=epositive, wrist=wpositive, fatherId=fReference[0]}
  [1902] = {x=-501.748, y=249.996, z=22, rx=-180, rz=179.853, shoulder=lefty, elbow=epositive, wrist=wpositive, fatherId=fReference[0]}
  [1903] = {x=-500.333, y=250, z=22, rx=180, rz=-179.947, shoulder=lefty, elbow=epositive, wrist=wpositive, fatherId=fReference[0]}
  [1904] = {x=-498.919, y=249.999, z=22, rx=-180, rz=-179.747, shoulder=lefty, elbow=epositive, wrist=wpositive, fatherId=fReference[0]}
  [1905] = {x=-497.504, y=249.992, z=22, rx=-180, rz=-179.547, shoulder=lefty, elbow=epositive, wrist=wpositive, fatherId=fReference[0]}
  [1906] = {x=-496.09, y=249.981, z=22, rx=-180, rz=-179.347, shoulder=lefty, elbow=epositive, wrist=wpositive, fatherId=fReference[0]}
  [1907] = {x=-494.676, y=249.965, z=22, rx=180, rz=-179.147, shoulder=lefty, elbow=epositive, wrist=wpositive, fatherId=fReference[0]}
  [1908] = {x=-493.261, y=249.944, z=22, rx=-180, rz=-178.947, shoulder=lefty, elbow=epositive, wrist=wpositive, fatherId=fReference[0]}
  [1909] = {x=-491.847, y=249.918, z=22, rx=-180, rz=-178.748, shoulder=lefty, elbow=epositive, wrist=wpositive, fatherId=fReference[0]}
  [1910] = {x=-490.433, y=249.887, z=22, rx=-180, rz=-178.548, shoulder=lefty, elbow=epositive, wrist=wpositive, fatherId=fReference[0]}
  [1911] = {x=-489.019, y=249.851, z=22, rx=180, rz=-178.348, shoulder=lefty, elbow=epositive, wrist=wpositive, fatherId=fReference[0]}
  [1912] = {x=-487.604, y=249.81, z=22, rx=-180, rz=-178.149, shoulder=lefty, elbow=epositive, wrist=wpositive, fatherId=fReference[0]}
  [1913] = {x=-486.19, y=249.765, z=22, rx=180, rz=-177.949, shoulder=lefty, elbow=epositive, wrist=wpositive, fatherId=fReference[0]}
  [1914] = {x=-484.776, y=249.714, z=22, rx=180, rz=-177.75, shoulder=lefty, elbow=epositive, wrist=wpositive, fatherId=fReference[0]}
  [1915] = {x=-483.363, y=249.659, z=22, rx=-180, rz=-177.551, shoulder=lefty, elbow=epositive, wrist=wpositive, fatherId=fReference[0]}
  [1916] = {x=-481.949, y=249.598, z=22, rx=-180, rz=-177.351, shoulder=lefty, elbow=epositive, wrist=wpositive, fatherId=fReference[0]}
  [1917] = {x=-480.535, y=249.533, z=22, rx=180, rz=-177.152, shoulder=lefty, elbow=epositive, wrist=wpositive, fatherId=fReference[0]}
  [1918] = {x=-479.122, y=249.462, z=22, rx=-180, rz=-176.954, shoulder=lefty, elbow=epositive, wrist=wpositive, fatherId=fReference[0]}
  [1919] = {x=-477.708, y=249.387, z=22, rx=180, rz=-176.755, shoulder=lefty, elbow=epositive, wrist=wpositive, fatherId=fReference[0]}
  [1920] = {x=-476.295, y=249.307, z=22, rx=-180, rz=-176.556, shoulder=lefty, elbow=epositive, wrist=wpositive, fatherId=fReference[0]}
  [1921] = {x=-474.882, y=249.222, z=22, rx=180, rz=-176.358, shoulder=lefty, elbow=epositive, wrist=wpositive, fatherId=fReference[0]}
  [1922] = {x=-473.469, y=249.132, z=22, rx=-180, rz=-176.16, shoulder=lefty, elbow=epositive, wrist=wpositive, fatherId=fReference[0]}
  [1923] = {x=-472.056, y=249.037, z=22, rx=-180, rz=-175.962, shoulder=lefty, elbow=epositive, wrist=wpositive, fatherId=fReference[0]}
  [1924] = {x=-470.643, y=248.937, z=22, rx=-180, rz=-175.764, shoulder=lefty, elbow=epositive, wrist=wpositive, fatherId=fReference[0]}
  [1925] = {x=-469.231, y=248.833, z=22, rx=180, rz=-175.566, shoulder=lefty, elbow=epositive, wrist=wpositive, fatherId=fReference[0]}
  [1926] = {x=-467.819, y=248.723, z=22, rx=-180, rz=-175.369, shoulder=lefty, elbow=epositive, wrist=wpositive, fatherId=fReference[0]}
  [1927] = {x=-466.407, y=248.609, z=22, rx=180, rz=-175.172, shoulder=lefty, elbow=epositive, wrist=wpositive, fatherId=fReference[0]}
  [1928] = {x=-464.995, y=248.49, z=22, rx=180, rz=-174.975, shoulder=lefty, elbow=epositive, wrist=wpositive, fatherId=fReference[0]}
  [1929] = {x=-463.583, y=248.366, z=22, rx=180, rz=-174.778, shoulder=lefty, elbow=epositive, wrist=wpositive, fatherId=fReference[0]}
  [1930] = {x=-462.172, y=248.237, z=22, rx=180, rz=-174.582, shoulder=lefty, elbow=epositive, wrist=wpositive, fatherId=fReference[0]}
  [1931] = {x=-460.76, y=248.103, z=22, rx=180, rz=-174.386, shoulder=lefty, elbow=epositive, wrist=wpositive, fatherId=fReference[0]}
  [1932] = {x=-459.349, y=247.964, z=22, rx=180, rz=-174.19, shoulder=lefty, elbow=epositive, wrist=wpositive, fatherId=fReference[0]}
  [1933] = {x=-457.939, y=247.82, z=22, rx=180, rz=-173.994, shoulder=lefty, elbow=epositive, wrist=wpositive, fatherId=fReference[0]}
  [1934] = {x=-456.528, y=247.672, z=22, rx=180, rz=-173.799, shoulder=lefty, elbow=epositive, wrist=wpositive, fatherId=fReference[0]}
  [1935] = {x=-455.118, y=247.519, z=22, rx=180, rz=-173.604, shoulder=lefty, elbow=epositive, wrist=wpositive, fatherId=fReference[0]}
  [1936] = {x=-453.708, y=247.361, z=22, rx=180, rz=-173.409, shoulder=lefty, elbow=epositive, wrist=wpositive, fatherId=fReference[0]}
  [1937] = {x=-452.298, y=247.198, z=22, rx=180, rz=-173.215, shoulder=lefty, elbow=epositive, wrist=wpositive, fatherId=fReference[0]}
  [1938] = {x=-450.889, y=247.03, z=22, rx=-180, rz=-173.021, shoulder=lefty, elbow=epositive, wrist=wpositive, fatherId=fReference[0]}
  [1939] = {x=-449.48, y=246.858, z=22, rx=-180, rz=-172.827, shoulder=lefty, elbow=epositive, wrist=wpositive, fatherId=fReference[0]}
  [1940] = {x=-448.071, y=246.68, z=22, rx=-180, rz=-172.634, shoulder=lefty, elbow=epositive, wrist=wpositive, fatherId=fReference[0]}
  [1941] = {x=-446.663, y=246.498, z=22, rx=-180, rz=-172.441, shoulder=lefty, elbow=epositive, wrist=wpositive, fatherId=fReference[0]}
  [1942] = {x=-445.254, y=246.312, z=22, rx=-180, rz=-172.248, shoulder=lefty, elbow=epositive, wrist=wpositive, fatherId=fReference[0]}
  [1943] = {x=-443.847, y=246.12, z=22, rx=180, rz=-172.056, shoulder=lefty, elbow=epositive, wrist=wpositive, fatherId=fReference[0]}
  [1944] = {x=-442.439, y=245.923, z=22, rx=-180, rz=-171.864, shoulder=lefty, elbow=epositive, wrist=wpositive, fatherId=fReference[0]}
  [1945] = {x=-441.032, y=245.722, z=22, rx=180, rz=-171.673, shoulder=lefty, elbow=epositive, wrist=wpositive, fatherId=fReference[0]}
  [1946] = {x=-439.625, y=245.516, z=22, rx=180, rz=-171.482, shoulder=lefty, elbow=epositive, wrist=wpositive, fatherId=fReference[0]}
  [1947] = {x=-438.218, y=245.306, z=22, rx=180, rz=-171.291, shoulder=lefty, elbow=epositive, wrist=wpositive, fatherId=fReference[0]}
  [1948] = {x=-436.812, y=245.09, z=22, rx=180, rz=-171.101, shoulder=lefty, elbow=epositive, wrist=wpositive, fatherId=fReference[0]}
  [1949] = {x=-435.406, y=244.87, z=22, rx=-180, rz=-170.911, shoulder=lefty, elbow=epositive, wrist=wpositive, fatherId=fReference[0]}
  [1950] = {x=-434.001, y=244.645, z=22, rx=-180, rz=-170.721, shoulder=lefty, elbow=epositive, wrist=wpositive, fatherId=fReference[0]}
  [1951] = {x=-432.596, y=244.416, z=22, rx=180, rz=-170.532, shoulder=lefty, elbow=epositive, wrist=wpositive, fatherId=fReference[0]}
  [1952] = {x=-431.191, y=244.182, z=22, rx=180, rz=-170.344, shoulder=lefty, elbow=epositive, wrist=wpositive, fatherId=fReference[0]}
  [1953] = {x=-429.787, y=243.943, z=22, rx=-180, rz=-170.156, shoulder=lefty, elbow=epositive, wrist=wpositive, fatherId=fReference[0]}
  [1954] = {x=-428.383, y=243.699, z=22, rx=180, rz=-169.968, shoulder=lefty, elbow=epositive, wrist=wpositive, fatherId=fReference[0]}
  [1955] = {x=-426.98, y=243.451, z=22, rx=-180, rz=-169.781, shoulder=lefty, elbow=epositive, wrist=wpositive, fatherId=fReference[0]}
  [1956] = {x=-425.577, y=243.198, z=22, rx=180, rz=-169.594, shoulder=lefty, elbow=epositive, wrist=wpositive, fatherId=fReference[0]}
  [1957] = {x=-424.174, y=242.94, z=22, rx=180, rz=-169.408, shoulder=lefty, elbow=epositive, wrist=wpositive, fatherId=fReference[0]}
  [1958] = {x=-422.772, y=242.678, z=22, rx=180, rz=-169.222, shoulder=lefty, elbow=epositive, wrist=wpositive, fatherId=fReference[0]}
  [1959] = {x=-421.37, y=242.411, z=22, rx=-180, rz=-169.037, shoulder=lefty, elbow=epositive, wrist=wpositive, fatherId=fReference[0]}
  [1960] = {x=-419.969, y=242.14, z=22, rx=180, rz=-168.852, shoulder=lefty, elbow=epositive, wrist=wpositive, fatherId=fReference[0]}
  [1961] = {x=-418.568, y=241.864, z=22, rx=-180, rz=-168.667, shoulder=lefty, elbow=epositive, wrist=wpositive, fatherId=fReference[0]}
  [1962] = {x=-417.167, y=241.583, z=22, rx=-180, rz=-168.484, shoulder=lefty, elbow=epositive, wrist=wpositive, fatherId=fReference[0]}
  [1963] = {x=-415.767, y=241.298, z=22, rx=180, rz=-168.3, shoulder=lefty, elbow=epositive, wrist=wpositive, fatherId=fReference[0]}
  [1964] = {x=-414.368, y=241.008, z=22, rx=180, rz=-168.118, shoulder=lefty, elbow=epositive, wrist=wpositive, fatherId=fReference[0]}
  [1965] = {x=-412.969, y=240.713, z=22, rx=-180, rz=-167.935, shoulder=lefty, elbow=epositive, wrist=wpositive, fatherId=fReference[0]}
  [1966] = {x=-411.57, y=240.415, z=22, rx=180, rz=-167.754, shoulder=lefty, elbow=epositive, wrist=wpositive, fatherId=fReference[0]}
  [1967] = {x=-410.172, y=240.111, z=22, rx=180, rz=-167.573, shoulder=lefty, elbow=epositive, wrist=wpositive, fatherId=fReference[0]}
  [1968] = {x=-408.775, y=239.803, z=22, rx=180, rz=-167.392, shoulder=lefty, elbow=epositive, wrist=wpositive, fatherId=fReference[0]}
  [1969] = {x=-407.378, y=239.491, z=22, rx=180, rz=-167.212, shoulder=lefty, elbow=epositive, wrist=wpositive, fatherId=fReference[0]}
  [1970] = {x=-405.981, y=239.174, z=22, rx=180, rz=-167.033, shoulder=lefty, elbow=epositive, wrist=wpositive, fatherId=fReference[0]}
  [1971] = {x=-404.585, y=238.852, z=22, rx=-180, rz=-166.854, shoulder=lefty, elbow=epositive, wrist=wpositive, fatherId=fReference[0]}
  [1972] = {x=-403.189, y=238.526, z=22, rx=180, rz=-166.675, shoulder=lefty, elbow=epositive, wrist=wpositive, fatherId=fReference[0]}
  [1973] = {x=-401.794, y=238.196, z=22, rx=-180, rz=-166.498, shoulder=lefty, elbow=epositive, wrist=wpositive, fatherId=fReference[0]}
  [1974] = {x=-400.4, y=237.861, z=22, rx=-180, rz=-166.32, shoulder=lefty, elbow=epositive, wrist=wpositive, fatherId=fReference[0]}
  [1975] = {x=-399.006, y=237.522, z=22, rx=-180, rz=-166.144, shoulder=lefty, elbow=epositive, wrist=wpositive, fatherId=fReference[0]}
  [1976] = {x=-397.613, y=237.178, z=22, rx=180, rz=-165.968, shoulder=lefty, elbow=epositive, wrist=wpositive, fatherId=fReference[0]}
  [1977] = {x=-396.22, y=236.83, z=22, rx=-180, rz=-165.792, shoulder=lefty, elbow=epositive, wrist=wpositive, fatherId=fReference[0]}
  [1978] = {x=-394.827, y=236.477, z=22, rx=180, rz=-165.618, shoulder=lefty, elbow=epositive, wrist=wpositive, fatherId=fReference[0]}
  [1979] = {x=-393.436, y=236.12, z=22, rx=180, rz=-165.443, shoulder=lefty, elbow=epositive, wrist=wpositive, fatherId=fReference[0]}
  [1980] = {x=-392.044, y=235.759, z=22, rx=180, rz=-165.27, shoulder=lefty, elbow=epositive, wrist=wpositive, fatherId=fReference[0]}
  [1981] = {x=-390.654, y=235.394, z=22, rx=-180, rz=-165.097, shoulder=lefty, elbow=epositive, wrist=wpositive, fatherId=fReference[0]}
  [1982] = {x=-389.264, y=235.024, z=22, rx=180, rz=-164.924, shoulder=lefty, elbow=epositive, wrist=wpositive, fatherId=fReference[0]}
  [1983] = {x=-387.874, y=234.649, z=22, rx=-180, rz=-164.753, shoulder=lefty, elbow=epositive, wrist=wpositive, fatherId=fReference[0]}
  [1984] = {x=-386.485, y=234.271, z=22, rx=-180, rz=-164.582, shoulder=lefty, elbow=epositive, wrist=wpositive, fatherId=fReference[0]}
  [1985] = {x=-385.097, y=233.888, z=22, rx=180, rz=-164.411, shoulder=lefty, elbow=epositive, wrist=wpositive, fatherId=fReference[0]}
  [1986] = {x=-383.709, y=233.501, z=22, rx=-180, rz=-164.241, shoulder=lefty, elbow=epositive, wrist=wpositive, fatherId=fReference[0]}
  [1987] = {x=-382.322, y=233.109, z=22, rx=180, rz=-164.072, shoulder=lefty, elbow=epositive, wrist=wpositive, fatherId=fReference[0]}
  [1988] = {x=-380.936, y=232.714, z=22, rx=180, rz=-163.904, shoulder=lefty, elbow=epositive, wrist=wpositive, fatherId=fReference[0]}
  [1989] = {x=-379.55, y=232.314, z=22, rx=-180, rz=-163.736, shoulder=lefty, elbow=epositive, wrist=wpositive, fatherId=fReference[0]}
  [1990] = {x=-378.164, y=231.909, z=22, rx=-180, rz=-163.568, shoulder=lefty, elbow=epositive, wrist=wpositive, fatherId=fReference[0]}
  [1991] = {x=-376.78, y=231.501, z=22, rx=180, rz=-163.402, shoulder=lefty, elbow=epositive, wrist=wpositive, fatherId=fReference[0]}
  [1992] = {x=-375.395, y=231.089, z=22, rx=180, rz=-163.236, shoulder=lefty, elbow=epositive, wrist=wpositive, fatherId=fReference[0]}
  [1993] = {x=-374.012, y=230.672, z=22, rx=180, rz=-163.071, shoulder=lefty, elbow=epositive, wrist=wpositive, fatherId=fReference[0]}
  [1994] = {x=-372.629, y=230.251, z=22, rx=-180, rz=-162.906, shoulder=lefty, elbow=epositive, wrist=wpositive, fatherId=fReference[0]}
  [1995] = {x=-371.247, y=229.826, z=22, rx=180, rz=-162.742, shoulder=lefty, elbow=epositive, wrist=wpositive, fatherId=fReference[0]}
  [1996] = {x=-369.865, y=229.397, z=22, rx=180, rz=-162.579, shoulder=lefty, elbow=epositive, wrist=wpositive, fatherId=fReference[0]}
  [1997] = {x=-368.484, y=228.963, z=22, rx=-180, rz=-162.416, shoulder=lefty, elbow=epositive, wrist=wpositive, fatherId=fReference[0]}
  [1998] = {x=-367.104, y=228.526, z=22, rx=180, rz=-162.254, shoulder=lefty, elbow=epositive, wrist=wpositive, fatherId=fReference[0]}
  [1999] = {x=-365.724, y=228.084, z=22, rx=-180, rz=-162.093, shoulder=lefty, elbow=epositive, wrist=wpositive, fatherId=fReference[0]}
  [2000] = {x=-364.345, y=227.639, z=22, rx=-180, rz=-161.932, shoulder=lefty, elbow=epositive, wrist=wpositive, fatherId=fReference[0]}
  [2001] = {x=-362.966, y=227.189, z=22, rx=180, rz=-161.772, shoulder=lefty, elbow=epositive, wrist=wpositive, fatherId=fReference[0]}
  [2002] = {x=-361.588, y=226.735, z=22, rx=180, rz=-161.613, shoulder=lefty, elbow=epositive, wrist=wpositive, fatherId=fReference[0]}
  [2003] = {x=-360.211, y=226.277, z=22, rx=-180, rz=-161.455, shoulder=lefty, elbow=epositive, wrist=wpositive, fatherId=fReference[0]}
  [2004] = {x=-358.835, y=225.816, z=22, rx=-180, rz=-161.297, shoulder=lefty, elbow=epositive, wrist=wpositive, fatherId=fReference[0]}
  [2005] = {x=-357.459, y=225.35, z=22, rx=-180, rz=-161.14, shoulder=lefty, elbow=epositive, wrist=wpositive, fatherId=fReference[0]}
  [2006] = {x=-356.084, y=224.88, z=22, rx=-180, rz=-160.983, shoulder=lefty, elbow=epositive, wrist=wpositive, fatherId=fReference[0]}
  [2007] = {x=-354.709, y=224.406, z=22, rx=-180, rz=-160.828, shoulder=lefty, elbow=epositive, wrist=wpositive, fatherId=fReference[0]}
  [2008] = {x=-353.335, y=223.929, z=22, rx=180, rz=-160.673, shoulder=lefty, elbow=epositive, wrist=wpositive, fatherId=fReference[0]}
  [2009] = {x=-351.962, y=223.447, z=22, rx=180, rz=-160.518, shoulder=lefty, elbow=epositive, wrist=wpositive, fatherId=fReference[0]}
  [2010] = {x=-350.59, y=222.961, z=22, rx=-180, rz=-160.365, shoulder=lefty, elbow=epositive, wrist=wpositive, fatherId=fReference[0]}
  [2011] = {x=-349.218, y=222.472, z=22, rx=-180, rz=-160.212, shoulder=lefty, elbow=epositive, wrist=wpositive, fatherId=fReference[0]}
  [2012] = {x=-347.847, y=221.979, z=22, rx=-180, rz=-160.06, shoulder=lefty, elbow=epositive, wrist=wpositive, fatherId=fReference[0]}
  [2013] = {x=-346.476, y=221.482, z=22, rx=-180, rz=-159.908, shoulder=lefty, elbow=epositive, wrist=wpositive, fatherId=fReference[0]}
  [2014] = {x=-345.107, y=220.98, z=22, rx=-180, rz=-159.757, shoulder=lefty, elbow=epositive, wrist=wpositive, fatherId=fReference[0]}
  [2015] = {x=-343.737, y=220.476, z=22, rx=-180, rz=-159.607, shoulder=lefty, elbow=epositive, wrist=wpositive, fatherId=fReference[0]}
  [2016] = {x=-342.369, y=219.967, z=22, rx=180, rz=-159.458, shoulder=lefty, elbow=epositive, wrist=wpositive, fatherId=fReference[0]}
  [2017] = {x=-341.001, y=219.454, z=22, rx=-180, rz=-159.309, shoulder=lefty, elbow=epositive, wrist=wpositive, fatherId=fReference[0]}
  [2018] = {x=-339.634, y=218.938, z=22, rx=-180, rz=-159.161, shoulder=lefty, elbow=epositive, wrist=wpositive, fatherId=fReference[0]}
  [2019] = {x=-338.268, y=218.418, z=22, rx=180, rz=-159.014, shoulder=lefty, elbow=epositive, wrist=wpositive, fatherId=fReference[0]}
  [2020] = {x=-336.903, y=217.894, z=22, rx=180, rz=-158.868, shoulder=lefty, elbow=epositive, wrist=wpositive, fatherId=fReference[0]}
  [2021] = {x=-335.538, y=217.367, z=22, rx=180, rz=-158.722, shoulder=lefty, elbow=epositive, wrist=wpositive, fatherId=fReference[0]}
  [2022] = {x=-334.173, y=216.835, z=22, rx=-180, rz=-158.577, shoulder=lefty, elbow=epositive, wrist=wpositive, fatherId=fReference[0]}
  [2023] = {x=-332.81, y=216.3, z=22, rx=180, rz=-158.433, shoulder=lefty, elbow=epositive, wrist=wpositive, fatherId=fReference[0]}
  [2024] = {x=-331.447, y=215.762, z=22, rx=180, rz=-158.289, shoulder=lefty, elbow=epositive, wrist=wpositive, fatherId=fReference[0]}
  [2025] = {x=-330.085, y=215.219, z=22, rx=-180, rz=-158.146, shoulder=lefty, elbow=epositive, wrist=wpositive, fatherId=fReference[0]}
  [2026] = {x=-328.724, y=214.674, z=22, rx=180, rz=-158.004, shoulder=lefty, elbow=epositive, wrist=wpositive, fatherId=fReference[0]}
  [2027] = {x=-327.363, y=214.124, z=22, rx=-180, rz=-157.862, shoulder=lefty, elbow=epositive, wrist=wpositive, fatherId=fReference[0]}
  [2028] = {x=-326.004, y=213.571, z=22, rx=-180, rz=-157.722, shoulder=lefty, elbow=epositive, wrist=wpositive, fatherId=fReference[0]}
  [2029] = {x=-324.644, y=213.014, z=22, rx=-180, rz=-157.582, shoulder=lefty, elbow=epositive, wrist=wpositive, fatherId=fReference[0]}
  [2030] = {x=-323.286, y=212.453, z=22, rx=-180, rz=-157.442, shoulder=lefty, elbow=epositive, wrist=wpositive, fatherId=fReference[0]}
  [2031] = {x=-321.928, y=211.89, z=22, rx=180, rz=-157.304, shoulder=lefty, elbow=epositive, wrist=wpositive, fatherId=fReference[0]}
  [2032] = {x=-320.571, y=211.322, z=22, rx=-180, rz=-157.166, shoulder=lefty, elbow=epositive, wrist=wpositive, fatherId=fReference[0]}
  [2033] = {x=-319.215, y=210.751, z=22, rx=180, rz=-157.029, shoulder=lefty, elbow=epositive, wrist=wpositive, fatherId=fReference[0]}
  [2034] = {x=-317.86, y=210.176, z=22, rx=-180, rz=-156.893, shoulder=lefty, elbow=epositive, wrist=wpositive, fatherId=fReference[0]}
  [2035] = {x=-316.505, y=209.598, z=22, rx=-180, rz=-156.757, shoulder=lefty, elbow=epositive, wrist=wpositive, fatherId=fReference[0]}
  [2036] = {x=-315.151, y=209.017, z=22, rx=180, rz=-156.622, shoulder=lefty, elbow=epositive, wrist=wpositive, fatherId=fReference[0]}
  [2037] = {x=-313.798, y=208.432, z=22, rx=180, rz=-156.488, shoulder=lefty, elbow=epositive, wrist=wpositive, fatherId=fReference[0]}
  [2038] = {x=-312.445, y=207.843, z=22, rx=-180, rz=-156.354, shoulder=lefty, elbow=epositive, wrist=wpositive, fatherId=fReference[0]}
  [2039] = {x=-311.094, y=207.252, z=22, rx=180, rz=-156.222, shoulder=lefty, elbow=epositive, wrist=wpositive, fatherId=fReference[0]}
  [2040] = {x=-309.743, y=206.656, z=22, rx=-180, rz=-156.09, shoulder=lefty, elbow=epositive, wrist=wpositive, fatherId=fReference[0]}
  [2041] = {x=-308.392, y=206.058, z=22, rx=-180, rz=-155.958, shoulder=lefty, elbow=epositive, wrist=wpositive, fatherId=fReference[0]}
  [2042] = {x=-307.043, y=205.456, z=22, rx=180, rz=-155.828, shoulder=lefty, elbow=epositive, wrist=wpositive, fatherId=fReference[0]}
  [2043] = {x=-305.694, y=204.85, z=22, rx=-180, rz=-155.698, shoulder=lefty, elbow=epositive, wrist=wpositive, fatherId=fReference[0]}
  [2044] = {x=-304.346, y=204.242, z=22, rx=180, rz=-155.569, shoulder=lefty, elbow=epositive, wrist=wpositive, fatherId=fReference[0]}
  [2045] = {x=-302.999, y=203.63, z=22, rx=-180, rz=-155.44, shoulder=lefty, elbow=epositive, wrist=wpositive, fatherId=fReference[0]}
  [2046] = {x=-301.652, y=203.014, z=22, rx=180, rz=-155.312, shoulder=lefty, elbow=epositive, wrist=wpositive, fatherId=fReference[0]}
  [2047] = {x=-300.307, y=202.396, z=22, rx=180, rz=-155.185, shoulder=lefty, elbow=epositive, wrist=wpositive, fatherId=fReference[0]}
  [2048] = {x=-298.962, y=201.774, z=22, rx=180, rz=-155.059, shoulder=lefty, elbow=epositive, wrist=wpositive, fatherId=fReference[0]}
  [2049] = {x=-297.618, y=201.149, z=22, rx=180, rz=-154.934, shoulder=lefty, elbow=epositive, wrist=wpositive, fatherId=fReference[0]}
  [2050] = {x=-296.274, y=200.52, z=22, rx=180, rz=-154.809, shoulder=lefty, elbow=epositive, wrist=wpositive, fatherId=fReference[0]}
  [2051] = {x=-294.931, y=199.889, z=22, rx=-180, rz=-154.685, shoulder=lefty, elbow=epositive, wrist=wpositive, fatherId=fReference[0]}
  [2052] = {x=-293.589, y=199.254, z=22, rx=180, rz=-154.561, shoulder=lefty, elbow=epositive, wrist=wpositive, fatherId=fReference[0]}
  [2053] = {x=-292.248, y=198.616, z=22, rx=-180, rz=-154.439, shoulder=lefty, elbow=epositive, wrist=wpositive, fatherId=fReference[0]}
  [2054] = {x=-290.908, y=197.975, z=22, rx=180, rz=-154.317, shoulder=lefty, elbow=epositive, wrist=wpositive, fatherId=fReference[0]}
  [2055] = {x=-289.568, y=197.331, z=22, rx=-180, rz=-154.195, shoulder=lefty, elbow=epositive, wrist=wpositive, fatherId=fReference[0]}
  [2056] = {x=-288.229, y=196.683, z=22, rx=180, rz=-154.075, shoulder=lefty, elbow=epositive, wrist=wpositive, fatherId=fReference[0]}
  [2057] = {x=-286.891, y=196.033, z=22, rx=-180, rz=-153.955, shoulder=lefty, elbow=epositive, wrist=wpositive, fatherId=fReference[0]}
  [2058] = {x=-285.554, y=195.379, z=22, rx=180, rz=-153.836, shoulder=lefty, elbow=epositive, wrist=wpositive, fatherId=fReference[0]}
  [2059] = {x=-284.217, y=194.723, z=22, rx=180, rz=-153.718, shoulder=lefty, elbow=epositive, wrist=wpositive, fatherId=fReference[0]}
  [2060] = {x=-282.882, y=194.063, z=22, rx=-180, rz=-153.6, shoulder=lefty, elbow=epositive, wrist=wpositive, fatherId=fReference[0]}
  [2061] = {x=-281.546, y=193.4, z=22, rx=-180, rz=-153.483, shoulder=lefty, elbow=epositive, wrist=wpositive, fatherId=fReference[0]}
  [2062] = {x=-280.212, y=192.734, z=22, rx=-180, rz=-153.367, shoulder=lefty, elbow=epositive, wrist=wpositive, fatherId=fReference[0]}
  [2063] = {x=-278.879, y=192.066, z=22, rx=180, rz=-153.251, shoulder=lefty, elbow=epositive, wrist=wpositive, fatherId=fReference[0]}
  [2064] = {x=-277.546, y=191.394, z=22, rx=-180, rz=-153.136, shoulder=lefty, elbow=epositive, wrist=wpositive, fatherId=fReference[0]}
  [2065] = {x=-276.214, y=190.719, z=22, rx=180, rz=-153.022, shoulder=lefty, elbow=epositive, wrist=wpositive, fatherId=fReference[0]}
  [2066] = {x=-274.883, y=190.042, z=22, rx=-180, rz=-152.908, shoulder=lefty, elbow=epositive, wrist=wpositive, fatherId=fReference[0]}
  [2067] = {x=-273.552, y=189.361, z=22, rx=180, rz=-152.796, shoulder=lefty, elbow=epositive, wrist=wpositive, fatherId=fReference[0]}
  [2068] = {x=-272.222, y=188.678, z=22, rx=-180, rz=-152.684, shoulder=lefty, elbow=epositive, wrist=wpositive, fatherId=fReference[0]}
  [2069] = {x=-270.894, y=187.991, z=22, rx=-180, rz=-152.572, shoulder=lefty, elbow=epositive, wrist=wpositive, fatherId=fReference[0]}
  [2070] = {x=-269.565, y=187.302, z=22, rx=180, rz=-152.461, shoulder=lefty, elbow=epositive, wrist=wpositive, fatherId=fReference[0]}
  [2071] = {x=-268.238, y=186.61, z=22, rx=180, rz=-152.351, shoulder=lefty, elbow=epositive, wrist=wpositive, fatherId=fReference[0]}
  [2072] = {x=-266.911, y=185.915, z=22, rx=180, rz=-152.242, shoulder=lefty, elbow=epositive, wrist=wpositive, fatherId=fReference[0]}
  [2073] = {x=-265.585, y=185.217, z=22, rx=180, rz=-152.134, shoulder=lefty, elbow=epositive, wrist=wpositive, fatherId=fReference[0]}
  [2074] = {x=-264.26, y=184.516, z=22, rx=-180, rz=-152.026, shoulder=lefty, elbow=epositive, wrist=wpositive, fatherId=fReference[0]}
  [2075] = {x=-262.936, y=183.813, z=22, rx=180, rz=-151.918, shoulder=lefty, elbow=epositive, wrist=wpositive, fatherId=fReference[0]}
  [2076] = {x=-261.612, y=183.107, z=22, rx=180, rz=-151.812, shoulder=lefty, elbow=epositive, wrist=wpositive, fatherId=fReference[0]}
  [2077] = {x=-260.289, y=182.398, z=22, rx=180, rz=-151.706, shoulder=lefty, elbow=epositive, wrist=wpositive, fatherId=fReference[0]}
  [2078] = {x=-258.967, y=181.686, z=22, rx=180, rz=-151.601, shoulder=lefty, elbow=epositive, wrist=wpositive, fatherId=fReference[0]}
  [2079] = {x=-257.646, y=180.972, z=22, rx=-180, rz=-151.496, shoulder=lefty, elbow=epositive, wrist=wpositive, fatherId=fReference[0]}
  [2080] = {x=-256.325, y=180.254, z=22, rx=180, rz=-151.392, shoulder=lefty, elbow=epositive, wrist=wpositive, fatherId=fReference[0]}
  [2081] = {x=-255.005, y=179.535, z=22, rx=-180, rz=-151.289, shoulder=lefty, elbow=epositive, wrist=wpositive, fatherId=fReference[0]}
  [2082] = {x=-253.686, y=178.812, z=22, rx=180, rz=-151.187, shoulder=lefty, elbow=epositive, wrist=wpositive, fatherId=fReference[0]}
  [2083] = {x=-252.368, y=178.087, z=22, rx=180, rz=-151.085, shoulder=lefty, elbow=epositive, wrist=wpositive, fatherId=fReference[0]}
  [2084] = {x=-251.05, y=177.359, z=22, rx=-180, rz=-150.984, shoulder=lefty, elbow=epositive, wrist=wpositive, fatherId=fReference[0]}
  [2085] = {x=-249.733, y=176.629, z=22, rx=-180, rz=-150.883, shoulder=lefty, elbow=epositive, wrist=wpositive, fatherId=fReference[0]}
  [2086] = {x=-248.417, y=175.895, z=22, rx=180, rz=-150.784, shoulder=lefty, elbow=epositive, wrist=wpositive, fatherId=fReference[0]}
  [2087] = {x=-247.102, y=175.16, z=22, rx=-180, rz=-150.685, shoulder=lefty, elbow=epositive, wrist=wpositive, fatherId=fReference[0]}
  [2088] = {x=-245.787, y=174.422, z=22, rx=-180, rz=-150.586, shoulder=lefty, elbow=epositive, wrist=wpositive, fatherId=fReference[0]}
  [2089] = {x=-244.473, y=173.681, z=22, rx=-180, rz=-150.488, shoulder=lefty, elbow=epositive, wrist=wpositive, fatherId=fReference[0]}
  [2090] = {x=-243.16, y=172.937, z=22, rx=180, rz=-150.391, shoulder=lefty, elbow=epositive, wrist=wpositive, fatherId=fReference[0]}
  [2091] = {x=-241.847, y=172.192, z=22, rx=180, rz=-150.295, shoulder=lefty, elbow=epositive, wrist=wpositive, fatherId=fReference[0]}
  [2092] = {x=-240.536, y=171.443, z=22, rx=-180, rz=-150.199, shoulder=lefty, elbow=epositive, wrist=wpositive, fatherId=fReference[0]}
  [2093] = {x=-239.225, y=170.692, z=22, rx=180, rz=-150.104, shoulder=lefty, elbow=epositive, wrist=wpositive, fatherId=fReference[0]}
  [2094] = {x=-237.914, y=169.939, z=22, rx=180, rz=-150.009, shoulder=lefty, elbow=epositive, wrist=wpositive, fatherId=fReference[0]}
  [2095] = {x=-236.605, y=169.183, z=22, rx=-180, rz=-149.915, shoulder=lefty, elbow=epositive, wrist=wpositive, fatherId=fReference[0]}
  [2096] = {x=-235.296, y=168.425, z=22, rx=-180, rz=-149.822, shoulder=lefty, elbow=epositive, wrist=wpositive, fatherId=fReference[0]}
  [2097] = {x=-233.988, y=167.664, z=22, rx=-180, rz=-149.729, shoulder=lefty, elbow=epositive, wrist=wpositive, fatherId=fReference[0]}
  [2098] = {x=-232.68, y=166.901, z=22, rx=180, rz=-149.638, shoulder=lefty, elbow=epositive, wrist=wpositive, fatherId=fReference[0]}
  [2099] = {x=-231.373, y=166.136, z=22, rx=-180, rz=-149.546, shoulder=lefty, elbow=epositive, wrist=wpositive, fatherId=fReference[0]}
  [2100] = {x=-230.067, y=165.368, z=22, rx=-180, rz=-149.456, shoulder=lefty, elbow=epositive, wrist=wpositive, fatherId=fReference[0]}
  [2101] = {x=-228.762, y=164.597, z=22, rx=-180, rz=-149.366, shoulder=lefty, elbow=epositive, wrist=wpositive, fatherId=fReference[0]}
  [2102] = {x=-227.457, y=163.825, z=22, rx=-180, rz=-149.276, shoulder=lefty, elbow=epositive, wrist=wpositive, fatherId=fReference[0]}
  [2103] = {x=-226.153, y=163.05, z=22, rx=180, rz=-149.187, shoulder=lefty, elbow=epositive, wrist=wpositive, fatherId=fReference[0]}
  [2104] = {x=-224.85, y=162.272, z=22, rx=180, rz=-149.099, shoulder=lefty, elbow=epositive, wrist=wpositive, fatherId=fReference[0]}
  [2105] = {x=-223.547, y=161.493, z=22, rx=180, rz=-149.012, shoulder=lefty, elbow=epositive, wrist=wpositive, fatherId=fReference[0]}
  [2106] = {x=-222.245, y=160.711, z=22, rx=-180, rz=-148.925, shoulder=lefty, elbow=epositive, wrist=wpositive, fatherId=fReference[0]}
  [2107] = {x=-220.944, y=159.927, z=22, rx=-180, rz=-148.839, shoulder=lefty, elbow=epositive, wrist=wpositive, fatherId=fReference[0]}
  [2108] = {x=-219.643, y=159.14, z=22, rx=180, rz=-148.753, shoulder=lefty, elbow=epositive, wrist=wpositive, fatherId=fReference[0]}
  [2109] = {x=-218.344, y=158.351, z=22, rx=-180, rz=-148.668, shoulder=lefty, elbow=epositive, wrist=wpositive, fatherId=fReference[0]}
  [2110] = {x=-217.044, y=157.56, z=22, rx=-180, rz=-148.584, shoulder=lefty, elbow=epositive, wrist=wpositive, fatherId=fReference[0]}
  [2111] = {x=-215.746, y=156.767, z=22, rx=180, rz=-148.5, shoulder=lefty, elbow=epositive, wrist=wpositive, fatherId=fReference[0]}
  [2112] = {x=-214.448, y=155.972, z=22, rx=-180, rz=-148.417, shoulder=lefty, elbow=epositive, wrist=wpositive, fatherId=fReference[0]}
  [2113] = {x=-213.15, y=155.174, z=22, rx=-180, rz=-148.334, shoulder=lefty, elbow=epositive, wrist=wpositive, fatherId=fReference[0]}
  [2114] = {x=-211.854, y=154.375, z=22, rx=180, rz=-148.252, shoulder=lefty, elbow=epositive, wrist=wpositive, fatherId=fReference[0]}
  [2115] = {x=-210.558, y=153.573, z=22, rx=180, rz=-148.171, shoulder=lefty, elbow=epositive, wrist=wpositive, fatherId=fReference[0]}
  [2116] = {x=-209.262, y=152.769, z=22, rx=-180, rz=-148.09, shoulder=lefty, elbow=epositive, wrist=wpositive, fatherId=fReference[0]}
  [2117] = {x=-207.968, y=151.962, z=22, rx=-180, rz=-148.01, shoulder=lefty, elbow=epositive, wrist=wpositive, fatherId=fReference[0]}
  [2118] = {x=-206.674, y=151.154, z=22, rx=-180, rz=-147.931, shoulder=lefty, elbow=epositive, wrist=wpositive, fatherId=fReference[0]}
  [2119] = {x=-205.38, y=150.344, z=22, rx=-180, rz=-147.852, shoulder=lefty, elbow=epositive, wrist=wpositive, fatherId=fReference[0]}
  [2120] = {x=-204.088, y=149.531, z=22, rx=180, rz=-147.774, shoulder=lefty, elbow=epositive, wrist=wpositive, fatherId=fReference[0]}
  [2121] = {x=-202.795, y=148.717, z=22, rx=-180, rz=-147.696, shoulder=lefty, elbow=epositive, wrist=wpositive, fatherId=fReference[0]}
  [2122] = {x=-201.504, y=147.9, z=22, rx=-180, rz=-147.619, shoulder=lefty, elbow=epositive, wrist=wpositive, fatherId=fReference[0]}
  [2123] = {x=-200.213, y=147.082, z=22, rx=180, rz=-147.542, shoulder=lefty, elbow=epositive, wrist=wpositive, fatherId=fReference[0]}
  [2124] = {x=-198.923, y=146.261, z=22, rx=-180, rz=-147.467, shoulder=lefty, elbow=epositive, wrist=wpositive, fatherId=fReference[0]}
  [2125] = {x=-197.633, y=145.438, z=22, rx=-180, rz=-147.391, shoulder=lefty, elbow=epositive, wrist=wpositive, fatherId=fReference[0]}
  [2126] = {x=-196.344, y=144.614, z=22, rx=180, rz=-147.317, shoulder=lefty, elbow=epositive, wrist=wpositive, fatherId=fReference[0]}
  [2127] = {x=-195.055, y=143.787, z=22, rx=180, rz=-147.242, shoulder=lefty, elbow=epositive, wrist=wpositive, fatherId=fReference[0]}
  [2128] = {x=-193.768, y=142.958, z=22, rx=-180, rz=-147.169, shoulder=lefty, elbow=epositive, wrist=wpositive, fatherId=fReference[0]}
  [2129] = {x=-192.48, y=142.128, z=22, rx=-180, rz=-147.096, shoulder=lefty, elbow=epositive, wrist=wpositive, fatherId=fReference[0]}
  [2130] = {x=-191.194, y=141.295, z=22, rx=-180, rz=-147.024, shoulder=lefty, elbow=epositive, wrist=wpositive, fatherId=fReference[0]}
  [2131] = {x=-189.908, y=140.461, z=22, rx=-180, rz=-146.952, shoulder=lefty, elbow=epositive, wrist=wpositive, fatherId=fReference[0]}
  [2132] = {x=-188.622, y=139.625, z=22, rx=180, rz=-146.88, shoulder=lefty, elbow=epositive, wrist=wpositive, fatherId=fReference[0]}
  [2133] = {x=-187.337, y=138.786, z=22, rx=180, rz=-146.81, shoulder=lefty, elbow=epositive, wrist=wpositive, fatherId=fReference[0]}
  [2134] = {x=-186.053, y=137.946, z=22, rx=180, rz=-146.74, shoulder=lefty, elbow=epositive, wrist=wpositive, fatherId=fReference[0]}
  [2135] = {x=-184.769, y=137.104, z=22, rx=-180, rz=-146.67, shoulder=lefty, elbow=epositive, wrist=wpositive, fatherId=fReference[0]}
  [2136] = {x=-183.486, y=136.26, z=22, rx=180, rz=-146.601, shoulder=lefty, elbow=epositive, wrist=wpositive, fatherId=fReference[0]}
  [2137] = {x=-182.204, y=135.415, z=22, rx=180, rz=-146.533, shoulder=lefty, elbow=epositive, wrist=wpositive, fatherId=fReference[0]}
  [2138] = {x=-180.922, y=134.567, z=22, rx=-180, rz=-146.465, shoulder=lefty, elbow=epositive, wrist=wpositive, fatherId=fReference[0]}
  [2139] = {x=-179.641, y=133.718, z=22, rx=180, rz=-146.398, shoulder=lefty, elbow=epositive, wrist=wpositive, fatherId=fReference[0]}
  [2140] = {x=-178.36, y=132.867, z=22, rx=180, rz=-146.331, shoulder=lefty, elbow=epositive, wrist=wpositive, fatherId=fReference[0]}
  [2141] = {x=-177.08, y=132.014, z=22, rx=180, rz=-146.265, shoulder=lefty, elbow=epositive, wrist=wpositive, fatherId=fReference[0]}
  [2142] = {x=-175.8, y=131.16, z=22, rx=-180, rz=-146.199, shoulder=lefty, elbow=epositive, wrist=wpositive, fatherId=fReference[0]}
  [2143] = {x=-174.521, y=130.304, z=22, rx=180, rz=-146.134, shoulder=lefty, elbow=epositive, wrist=wpositive, fatherId=fReference[0]}
  [2144] = {x=-173.242, y=129.446, z=22, rx=-180, rz=-146.07, shoulder=lefty, elbow=epositive, wrist=wpositive, fatherId=fReference[0]}
  [2145] = {x=-171.964, y=128.586, z=22, rx=180, rz=-146.006, shoulder=lefty, elbow=epositive, wrist=wpositive, fatherId=fReference[0]}
  [2146] = {x=-170.687, y=127.724, z=22, rx=180, rz=-145.943, shoulder=lefty, elbow=epositive, wrist=wpositive, fatherId=fReference[0]}
  [2147] = {x=-169.41, y=126.861, z=22, rx=180, rz=-145.88, shoulder=lefty, elbow=epositive, wrist=wpositive, fatherId=fReference[0]}
  [2148] = {x=-168.134, y=125.996, z=22, rx=180, rz=-145.818, shoulder=lefty, elbow=epositive, wrist=wpositive, fatherId=fReference[0]}
  [2149] = {x=-166.858, y=125.13, z=22, rx=180, rz=-145.756, shoulder=lefty, elbow=epositive, wrist=wpositive, fatherId=fReference[0]}
  [2150] = {x=-165.583, y=124.262, z=22, rx=180, rz=-145.695, shoulder=lefty, elbow=epositive, wrist=wpositive, fatherId=fReference[0]}
  [2151] = {x=-164.308, y=123.392, z=22, rx=180, rz=-145.634, shoulder=lefty, elbow=epositive, wrist=wpositive, fatherId=fReference[0]}
  [2152] = {x=-163.034, y=122.521, z=22, rx=180, rz=-145.574, shoulder=lefty, elbow=epositive, wrist=wpositive, fatherId=fReference[0]}
  [2153] = {x=-161.76, y=121.648, z=22, rx=180, rz=-145.515, shoulder=lefty, elbow=epositive, wrist=wpositive, fatherId=fReference[0]}
  [2154] = {x=-160.487, y=120.773, z=22, rx=-180, rz=-145.455, shoulder=lefty, elbow=epositive, wrist=wpositive, fatherId=fReference[0]}
  [2155] = {x=-159.215, y=119.897, z=22, rx=180, rz=-145.397, shoulder=lefty, elbow=epositive, wrist=wpositive, fatherId=fReference[0]}
  [2156] = {x=-157.942, y=119.02, z=22, rx=-180, rz=-145.339, shoulder=lefty, elbow=epositive, wrist=wpositive, fatherId=fReference[0]}
  [2157] = {x=-156.671, y=118.141, z=22, rx=-180, rz=-145.282, shoulder=lefty, elbow=epositive, wrist=wpositive, fatherId=fReference[0]}
  [2158] = {x=-155.4, y=117.26, z=22, rx=180, rz=-145.225, shoulder=lefty, elbow=epositive, wrist=wpositive, fatherId=fReference[0]}
  [2159] = {x=-154.129, y=116.378, z=22, rx=180, rz=-145.168, shoulder=lefty, elbow=epositive, wrist=wpositive, fatherId=fReference[0]}
  [2160] = {x=-152.859, y=115.494, z=22, rx=180, rz=-145.113, shoulder=lefty, elbow=epositive, wrist=wpositive, fatherId=fReference[0]}
  [2161] = {x=-151.59, y=114.609, z=22, rx=180, rz=-145.057, shoulder=lefty, elbow=epositive, wrist=wpositive, fatherId=fReference[0]}
  [2162] = {x=-150.321, y=113.722, z=22, rx=-180, rz=-145.002, shoulder=lefty, elbow=epositive, wrist=wpositive, fatherId=fReference[0]}
  [2163] = {x=-149.052, y=112.834, z=22, rx=180, rz=-144.948, shoulder=lefty, elbow=epositive, wrist=wpositive, fatherId=fReference[0]}
  [2164] = {x=-147.784, y=111.944, z=22, rx=-180, rz=-144.894, shoulder=lefty, elbow=epositive, wrist=wpositive, fatherId=fReference[0]}
  [2165] = {x=-146.517, y=111.053, z=22, rx=-180, rz=-144.841, shoulder=lefty, elbow=epositive, wrist=wpositive, fatherId=fReference[0]}
  [2166] = {x=-145.25, y=110.161, z=22, rx=-180, rz=-144.789, shoulder=lefty, elbow=epositive, wrist=wpositive, fatherId=fReference[0]}
  [2167] = {x=-143.983, y=109.267, z=22, rx=180, rz=-144.736, shoulder=lefty, elbow=epositive, wrist=wpositive, fatherId=fReference[0]}
  [2168] = {x=-142.717, y=108.372, z=22, rx=-180, rz=-144.685, shoulder=lefty, elbow=epositive, wrist=wpositive, fatherId=fReference[0]}
  [2169] = {x=-141.452, y=107.475, z=22, rx=180, rz=-144.634, shoulder=lefty, elbow=epositive, wrist=wpositive, fatherId=fReference[0]}
  [2170] = {x=-140.187, y=106.578, z=22, rx=180, rz=-144.583, shoulder=lefty, elbow=epositive, wrist=wpositive, fatherId=fReference[0]}
  [2171] = {x=-138.922, y=105.678, z=22, rx=-180, rz=-144.533, shoulder=lefty, elbow=epositive, wrist=wpositive, fatherId=fReference[0]}
  [2172] = {x=-137.658, y=104.778, z=22, rx=180, rz=-144.483, shoulder=lefty, elbow=epositive, wrist=wpositive, fatherId=fReference[0]}
  [2173] = {x=-136.395, y=103.876, z=22, rx=-180, rz=-144.434, shoulder=lefty, elbow=epositive, wrist=wpositive, fatherId=fReference[0]}
  [2174] = {x=-135.131, y=102.973, z=22, rx=-180, rz=-144.385, shoulder=lefty, elbow=epositive, wrist=wpositive, fatherId=fReference[0]}
  [2175] = {x=-133.869, y=102.068, z=22, rx=-180, rz=-144.337, shoulder=lefty, elbow=epositive, wrist=wpositive, fatherId=fReference[0]}
  [2176] = {x=-132.606, y=101.162, z=22, rx=180, rz=-144.29, shoulder=lefty, elbow=epositive, wrist=wpositive, fatherId=fReference[0]}
  [2177] = {x=-131.345, y=100.255, z=22, rx=180, rz=-144.242, shoulder=lefty, elbow=epositive, wrist=wpositive, fatherId=fReference[0]}
  [2178] = {x=-130.083, y=99.347, z=22, rx=-180, rz=-144.196, shoulder=lefty, elbow=epositive, wrist=wpositive, fatherId=fReference[0]}
  [2179] = {x=-128.822, y=98.437, z=22, rx=-180, rz=-144.15, shoulder=lefty, elbow=epositive, wrist=wpositive, fatherId=fReference[0]}
  [2180] = {x=-127.562, y=97.527, z=22, rx=-180, rz=-144.104, shoulder=lefty, elbow=epositive, wrist=wpositive, fatherId=fReference[0]}
  [2181] = {x=-126.302, y=96.615, z=22, rx=180, rz=-144.059, shoulder=lefty, elbow=epositive, wrist=wpositive, fatherId=fReference[0]}
  [2182] = {x=-125.042, y=95.702, z=22, rx=-180, rz=-144.014, shoulder=lefty, elbow=epositive, wrist=wpositive, fatherId=fReference[0]}
  [2183] = {x=-123.783, y=94.787, z=22, rx=180, rz=-143.97, shoulder=lefty, elbow=epositive, wrist=wpositive, fatherId=fReference[0]}
  [2184] = {x=-122.525, y=93.872, z=22, rx=-180, rz=-143.926, shoulder=lefty, elbow=epositive, wrist=wpositive, fatherId=fReference[0]}
  [2185] = {x=-121.266, y=92.955, z=22, rx=-180, rz=-143.883, shoulder=lefty, elbow=epositive, wrist=wpositive, fatherId=fReference[0]}
  [2186] = {x=-120.009, y=92.037, z=22, rx=-180, rz=-143.841, shoulder=lefty, elbow=epositive, wrist=wpositive, fatherId=fReference[0]}
  [2187] = {x=-118.751, y=91.118, z=22, rx=180, rz=-143.798, shoulder=lefty, elbow=epositive, wrist=wpositive, fatherId=fReference[0]}
  [2188] = {x=-117.494, y=90.198, z=22, rx=-180, rz=-143.757, shoulder=lefty, elbow=epositive, wrist=wpositive, fatherId=fReference[0]}
  [2189] = {x=-116.238, y=89.277, z=22, rx=-180, rz=-143.715, shoulder=lefty, elbow=epositive, wrist=wpositive, fatherId=fReference[0]}
  [2190] = {x=-114.981, y=88.355, z=22, rx=-180, rz=-143.675, shoulder=lefty, elbow=epositive, wrist=wpositive, fatherId=fReference[0]}
  [2191] = {x=-113.726, y=87.432, z=22, rx=-180, rz=-143.634, shoulder=lefty, elbow=epositive, wrist=wpositive, fatherId=fReference[0]}
  [2192] = {x=-112.47, y=86.507, z=22, rx=180, rz=-143.595, shoulder=lefty, elbow=epositive, wrist=wpositive, fatherId=fReference[0]}
  [2193] = {x=-111.215, y=85.582, z=22, rx=-180, rz=-143.555, shoulder=lefty, elbow=epositive, wrist=wpositive, fatherId=fReference[0]}
  [2194] = {x=-109.961, y=84.656, z=22, rx=-180, rz=-143.516, shoulder=lefty, elbow=epositive, wrist=wpositive, fatherId=fReference[0]}
  [2195] = {x=-108.707, y=83.728, z=22, rx=-180, rz=-143.478, shoulder=lefty, elbow=epositive, wrist=wpositive, fatherId=fReference[0]}
  [2196] = {x=-107.453, y=82.8, z=22, rx=-180, rz=-143.44, shoulder=lefty, elbow=epositive, wrist=wpositive, fatherId=fReference[0]}
  [2197] = {x=-106.2, y=81.87, z=22, rx=-180, rz=-143.403, shoulder=lefty, elbow=epositive, wrist=wpositive, fatherId=fReference[0]}
  [2198] = {x=-104.947, y=80.94, z=22, rx=-180, rz=-143.366, shoulder=lefty, elbow=epositive, wrist=wpositive, fatherId=fReference[0]}
  [2199] = {x=-103.694, y=80.008, z=22, rx=-180, rz=-143.329, shoulder=lefty, elbow=epositive, wrist=wpositive, fatherId=fReference[0]}
  [2200] = {x=-102.442, y=79.076, z=22, rx=-180, rz=-143.293, shoulder=lefty, elbow=epositive, wrist=wpositive, fatherId=fReference[0]}
  [2201] = {x=-101.19, y=78.143, z=22, rx=-180, rz=-143.258, shoulder=lefty, elbow=epositive, wrist=wpositive, fatherId=fReference[0]}
  [2202] = {x=-99.938, y=77.208, z=22, rx=-180, rz=-143.223, shoulder=lefty, elbow=epositive, wrist=wpositive, fatherId=fReference[0]}
  [2203] = {x=-98.687, y=76.273, z=22, rx=-180, rz=-143.188, shoulder=lefty, elbow=epositive, wrist=wpositive, fatherId=fReference[0]}
  [2204] = {x=-97.437, y=75.337, z=22, rx=-180, rz=-143.154, shoulder=lefty, elbow=epositive, wrist=wpositive, fatherId=fReference[0]}
  [2205] = {x=-96.186, y=74.4, z=22, rx=180, rz=-143.12, shoulder=lefty, elbow=epositive, wrist=wpositive, fatherId=fReference[0]}
  [2206] = {x=-94.936, y=73.462, z=22, rx=-180, rz=-143.087, shoulder=lefty, elbow=epositive, wrist=wpositive, fatherId=fReference[0]}
  [2207] = {x=-93.686, y=72.523, z=22, rx=-180, rz=-143.054, shoulder=lefty, elbow=epositive, wrist=wpositive, fatherId=fReference[0]}
  [2208] = {x=-92.437, y=71.584, z=22, rx=-180, rz=-143.022, shoulder=lefty, elbow=epositive, wrist=wpositive, fatherId=fReference[0]}
  [2209] = {x=-91.188, y=70.643, z=22, rx=-180, rz=-142.99, shoulder=lefty, elbow=epositive, wrist=wpositive, fatherId=fReference[0]}
  [2210] = {x=-89.939, y=69.702, z=22, rx=-180, rz=-142.959, shoulder=lefty, elbow=epositive, wrist=wpositive, fatherId=fReference[0]}
  [2211] = {x=-88.691, y=68.76, z=22, rx=-180, rz=-142.928, shoulder=lefty, elbow=epositive, wrist=wpositive, fatherId=fReference[0]}
  [2212] = {x=-87.443, y=67.817, z=22, rx=-180, rz=-142.897, shoulder=lefty, elbow=epositive, wrist=wpositive, fatherId=fReference[0]}
  [2213] = {x=-86.195, y=66.873, z=22, rx=-180, rz=-142.867, shoulder=lefty, elbow=epositive, wrist=wpositive, fatherId=fReference[0]}
  [2214] = {x=-84.948, y=65.929, z=22, rx=180, rz=-142.838, shoulder=lefty, elbow=epositive, wrist=wpositive, fatherId=fReference[0]}
  [2215] = {x=-83.701, y=64.984, z=22, rx=180, rz=-142.809, shoulder=lefty, elbow=epositive, wrist=wpositive, fatherId=fReference[0]}
  [2216] = {x=-82.454, y=64.038, z=22, rx=-180, rz=-142.78, shoulder=lefty, elbow=epositive, wrist=wpositive, fatherId=fReference[0]}
  [2217] = {x=-81.208, y=63.091, z=22, rx=-180, rz=-142.752, shoulder=lefty, elbow=epositive, wrist=wpositive, fatherId=fReference[0]}
  [2218] = {x=-79.962, y=62.143, z=22, rx=180, rz=-142.724, shoulder=lefty, elbow=epositive, wrist=wpositive, fatherId=fReference[0]}
  [2219] = {x=-78.716, y=61.195, z=22, rx=-180, rz=-142.697, shoulder=lefty, elbow=epositive, wrist=wpositive, fatherId=fReference[0]}
  [2220] = {x=-77.47, y=60.246, z=22, rx=-180, rz=-142.67, shoulder=lefty, elbow=epositive, wrist=wpositive, fatherId=fReference[0]}
  [2221] = {x=-76.225, y=59.297, z=22, rx=-180, rz=-142.644, shoulder=lefty, elbow=epositive, wrist=wpositive, fatherId=fReference[0]}
  [2222] = {x=-74.98, y=58.346, z=22, rx=-180, rz=-142.618, shoulder=lefty, elbow=epositive, wrist=wpositive, fatherId=fReference[0]}
  [2223] = {x=-73.736, y=57.395, z=22, rx=180, rz=-142.592, shoulder=lefty, elbow=epositive, wrist=wpositive, fatherId=fReference[0]}
  [2224] = {x=-72.491, y=56.444, z=22, rx=-180, rz=-142.567, shoulder=lefty, elbow=epositive, wrist=wpositive, fatherId=fReference[0]}
  [2225] = {x=-71.247, y=55.491, z=22, rx=180, rz=-142.543, shoulder=lefty, elbow=epositive, wrist=wpositive, fatherId=fReference[0]}
  [2226] = {x=-70.003, y=54.538, z=22, rx=180, rz=-142.518, shoulder=lefty, elbow=epositive, wrist=wpositive, fatherId=fReference[0]}
  [2227] = {x=-68.76, y=53.585, z=22, rx=180, rz=-142.495, shoulder=lefty, elbow=epositive, wrist=wpositive, fatherId=fReference[0]}
  [2228] = {x=-67.516, y=52.63, z=22, rx=-180, rz=-142.471, shoulder=lefty, elbow=epositive, wrist=wpositive, fatherId=fReference[0]}
  [2229] = {x=-66.273, y=51.676, z=22, rx=180, rz=-142.449, shoulder=lefty, elbow=epositive, wrist=wpositive, fatherId=fReference[0]}
  [2230] = {x=-65.03, y=50.72, z=22, rx=-180, rz=-142.426, shoulder=lefty, elbow=epositive, wrist=wpositive, fatherId=fReference[0]}
  [2231] = {x=-63.788, y=49.764, z=22, rx=-180, rz=-142.404, shoulder=lefty, elbow=epositive, wrist=wpositive, fatherId=fReference[0]}
  [2232] = {x=-62.545, y=48.808, z=22, rx=-180, rz=-142.383, shoulder=lefty, elbow=epositive, wrist=wpositive, fatherId=fReference[0]}
  [2233] = {x=-61.303, y=47.85, z=22, rx=-180, rz=-142.362, shoulder=lefty, elbow=epositive, wrist=wpositive, fatherId=fReference[0]}
  [2234] = {x=-60.061, y=46.893, z=22, rx=-180, rz=-142.341, shoulder=lefty, elbow=epositive, wrist=wpositive, fatherId=fReference[0]}
  [2235] = {x=-58.82, y=45.934, z=22, rx=-180, rz=-142.321, shoulder=lefty, elbow=epositive, wrist=wpositive, fatherId=fReference[0]}
  [2236] = {x=-57.578, y=44.976, z=22, rx=-180, rz=-142.301, shoulder=lefty, elbow=epositive, wrist=wpositive, fatherId=fReference[0]}
  [2237] = {x=-56.337, y=44.016, z=22, rx=-180, rz=-142.282, shoulder=lefty, elbow=epositive, wrist=wpositive, fatherId=fReference[0]}
  [2238] = {x=-55.096, y=43.057, z=22, rx=180, rz=-142.263, shoulder=lefty, elbow=epositive, wrist=wpositive, fatherId=fReference[0]}
  [2239] = {x=-53.855, y=42.096, z=22, rx=180, rz=-142.244, shoulder=lefty, elbow=epositive, wrist=wpositive, fatherId=fReference[0]}
  [2240] = {x=-52.615, y=41.135, z=22, rx=-180, rz=-142.226, shoulder=lefty, elbow=epositive, wrist=wpositive, fatherId=fReference[0]}
  [2241] = {x=-51.374, y=40.174, z=22, rx=-180, rz=-142.209, shoulder=lefty, elbow=epositive, wrist=wpositive, fatherId=fReference[0]}
  [2242] = {x=-50.134, y=39.212, z=22, rx=-180, rz=-142.192, shoulder=lefty, elbow=epositive, wrist=wpositive, fatherId=fReference[0]}
  [2243] = {x=-48.894, y=38.25, z=22, rx=180, rz=-142.175, shoulder=lefty, elbow=epositive, wrist=wpositive, fatherId=fReference[0]}
  [2244] = {x=-47.654, y=37.288, z=22, rx=180, rz=-142.159, shoulder=lefty, elbow=epositive, wrist=wpositive, fatherId=fReference[0]}
  [2245] = {x=-46.414, y=36.325, z=22, rx=180, rz=-142.143, shoulder=lefty, elbow=epositive, wrist=wpositive, fatherId=fReference[0]}
  [2246] = {x=-45.175, y=35.361, z=22, rx=-180, rz=-142.127, shoulder=lefty, elbow=epositive, wrist=wpositive, fatherId=fReference[0]}
  [2247] = {x=-43.935, y=34.397, z=22, rx=-180, rz=-142.112, shoulder=lefty, elbow=epositive, wrist=wpositive, fatherId=fReference[0]}
  [2248] = {x=-42.696, y=33.433, z=22, rx=-180, rz=-142.098, shoulder=lefty, elbow=epositive, wrist=wpositive, fatherId=fReference[0]}
  [2249] = {x=-41.457, y=32.468, z=22, rx=-180, rz=-142.083, shoulder=lefty, elbow=epositive, wrist=wpositive, fatherId=fReference[0]}
  [2250] = {x=-40.218, y=31.503, z=22, rx=180, rz=-142.07, shoulder=lefty, elbow=epositive, wrist=wpositive, fatherId=fReference[0]}
  [2251] = {x=-38.979, y=30.538, z=22, rx=180, rz=-142.056, shoulder=lefty, elbow=epositive, wrist=wpositive, fatherId=fReference[0]}
  [2252] = {x=-37.74, y=29.572, z=22, rx=-180, rz=-142.044, shoulder=lefty, elbow=epositive, wrist=wpositive, fatherId=fReference[0]}
  [2253] = {x=-36.502, y=28.606, z=22, rx=-180, rz=-142.031, shoulder=lefty, elbow=epositive, wrist=wpositive, fatherId=fReference[0]}
  [2254] = {x=-35.263, y=27.639, z=22, rx=-180, rz=-142.019, shoulder=lefty, elbow=epositive, wrist=wpositive, fatherId=fReference[0]}
  [2255] = {x=-34.025, y=26.672, z=22, rx=-180, rz=-142.007, shoulder=lefty, elbow=epositive, wrist=wpositive, fatherId=fReference[0]}
  [2256] = {x=-32.787, y=25.705, z=22, rx=-180, rz=-141.996, shoulder=lefty, elbow=epositive, wrist=wpositive, fatherId=fReference[0]}
  [2257] = {x=-31.549, y=24.738, z=22, rx=-180, rz=-141.985, shoulder=lefty, elbow=epositive, wrist=wpositive, fatherId=fReference[0]}
  [2258] = {x=-30.311, y=23.77, z=22, rx=-180, rz=-141.975, shoulder=lefty, elbow=epositive, wrist=wpositive, fatherId=fReference[0]}
  [2259] = {x=-29.073, y=22.802, z=22, rx=-180, rz=-141.965, shoulder=lefty, elbow=epositive, wrist=wpositive, fatherId=fReference[0]}
  [2260] = {x=-27.835, y=21.834, z=22, rx=-180, rz=-141.956, shoulder=lefty, elbow=epositive, wrist=wpositive, fatherId=fReference[0]}
  [2261] = {x=-26.597, y=20.865, z=22, rx=180, rz=-141.947, shoulder=lefty, elbow=epositive, wrist=wpositive, fatherId=fReference[0]}
  [2262] = {x=-25.36, y=19.896, z=22, rx=-180, rz=-141.938, shoulder=lefty, elbow=epositive, wrist=wpositive, fatherId=fReference[0]}
  [2263] = {x=-24.122, y=18.927, z=22, rx=-180, rz=-141.93, shoulder=lefty, elbow=epositive, wrist=wpositive, fatherId=fReference[0]}
  [2264] = {x=-22.885, y=17.958, z=22, rx=-180, rz=-141.922, shoulder=lefty, elbow=epositive, wrist=wpositive, fatherId=fReference[0]}
  [2265] = {x=-21.647, y=16.988, z=22, rx=-180, rz=-141.915, shoulder=lefty, elbow=epositive, wrist=wpositive, fatherId=fReference[0]}
  [2266] = {x=-20.41, y=16.019, z=22, rx=-180, rz=-141.908, shoulder=lefty, elbow=epositive, wrist=wpositive, fatherId=fReference[0]}
  [2267] = {x=-19.172, y=15.049, z=22, rx=180, rz=-141.901, shoulder=lefty, elbow=epositive, wrist=wpositive, fatherId=fReference[0]}
  [2268] = {x=-17.935, y=14.079, z=22, rx=180, rz=-141.895, shoulder=lefty, elbow=epositive, wrist=wpositive, fatherId=fReference[0]}
  [2269] = {x=-16.698, y=13.109, z=22, rx=-180, rz=-141.889, shoulder=lefty, elbow=epositive, wrist=wpositive, fatherId=fReference[0]}
  [2270] = {x=-15.461, y=12.138, z=22, rx=-180, rz=-141.884, shoulder=lefty, elbow=epositive, wrist=wpositive, fatherId=fReference[0]}
  [2271] = {x=-14.224, y=11.168, z=22, rx=-180, rz=-141.879, shoulder=lefty, elbow=epositive, wrist=wpositive, fatherId=fReference[0]}
  [2272] = {x=-12.987, y=10.197, z=22, rx=180, rz=-141.875, shoulder=lefty, elbow=epositive, wrist=wpositive, fatherId=fReference[0]}
  [2273] = {x=-11.75, y=9.226, z=22, rx=-180, rz=-141.871, shoulder=lefty, elbow=epositive, wrist=wpositive, fatherId=fReference[0]}
  [2274] = {x=-10.513, y=8.255, z=22, rx=180, rz=-141.867, shoulder=lefty, elbow=epositive, wrist=wpositive, fatherId=fReference[0]}
  [2275] = {x=-9.276, y=7.284, z=22, rx=180, rz=-141.864, shoulder=lefty, elbow=epositive, wrist=wpositive, fatherId=fReference[0]}
  [2276] = {x=-8.039, y=6.313, z=22, rx=180, rz=-141.862, shoulder=lefty, elbow=epositive, wrist=wpositive, fatherId=fReference[0]}
  [2277] = {x=-6.802, y=5.342, z=22, rx=-180, rz=-141.859, shoulder=lefty, elbow=epositive, wrist=wpositive, fatherId=fReference[0]}
  [2278] = {x=-5.565, y=4.37, z=22, rx=-180, rz=-141.857, shoulder=lefty, elbow=epositive, wrist=wpositive, fatherId=fReference[0]}
  [2279] = {x=-4.328, y=3.399, z=22, rx=-180, rz=-141.856, shoulder=lefty, elbow=epositive, wrist=wpositive, fatherId=fReference[0]}
  [2280] = {x=-3.091, y=2.427, z=22, rx=180, rz=-141.855, shoulder=lefty, elbow=epositive, wrist=wpositive, fatherId=fReference[0]}
  [2281] = {x=-1.854, y=1.456, z=22, rx=-180, rz=-141.854, shoulder=lefty, elbow=epositive, wrist=wpositive, fatherId=fReference[0]}
  [2282] = {x=-0.617, y=0.484, z=22, rx=-180, rz=-141.854, shoulder=lefty, elbow=epositive, wrist=wpositive, fatherId=fReference[0]}
  [2283] = {x=0.62, y=-0.487, z=22, rx=-180, rz=-141.854, shoulder=lefty, elbow=epositive, wrist=wpositive, fatherId=fReference[0]}
  [2284] = {x=1.857, y=-1.459, z=22, rx=180, rz=-141.855, shoulder=lefty, elbow=epositive, wrist=wpositive, fatherId=fReference[0]}
  [2285] = {x=3.094, y=-2.43, z=22, rx=-180, rz=-141.856, shoulder=lefty, elbow=epositive, wrist=wpositive, fatherId=fReference[0]}
  [2286] = {x=4.331, y=-3.402, z=22, rx=180, rz=-141.857, shoulder=lefty, elbow=epositive, wrist=wpositive, fatherId=fReference[0]}
  [2287] = {x=5.568, y=-4.373, z=22, rx=180, rz=-141.859, shoulder=lefty, elbow=epositive, wrist=wpositive, fatherId=fReference[0]}
  [2288] = {x=6.805, y=-5.345, z=22, rx=180, rz=-141.862, shoulder=lefty, elbow=epositive, wrist=wpositive, fatherId=fReference[0]}
  [2289] = {x=8.043, y=-6.316, z=22, rx=-180, rz=-141.864, shoulder=lefty, elbow=epositive, wrist=wpositive, fatherId=fReference[0]}
  [2290] = {x=9.28, y=-7.287, z=22, rx=180, rz=-141.867, shoulder=lefty, elbow=epositive, wrist=wpositive, fatherId=fReference[0]}
  [2291] = {x=10.517, y=-8.259, z=22, rx=-180, rz=-141.871, shoulder=lefty, elbow=epositive, wrist=wpositive, fatherId=fReference[0]}
  [2292] = {x=11.754, y=-9.23, z=22, rx=180, rz=-141.875, shoulder=lefty, elbow=epositive, wrist=wpositive, fatherId=fReference[0]}
